LIN {X 0,Y 573.255,Z 289.769,A -85,B 0,C 180,E1 -2241.895,E2 -2241.895} C_VEL
LIN {X 0,Y 573.193,Z 298.434,A -85,B 0,C 180,E1 -2242.603,E2 -2242.603} C_VEL
LIN {X 0,Y 573.151,Z 305.582,A -85,B 0,C 180,E1 -2243.326,E2 -2243.326} C_VEL
LIN {X 0,Y 573.113,Z 312.436,A -85,B 0,C 180,E1 -2244.194,E2 -2244.194} C_VEL
LIN {X 0,Y 572.995,Z 317.989,A -85,B 0,C 180,E1 -2245.075,E2 -2245.075} C_VEL
LIN {X 0,Y 573.036,Z 323.15,A -85,B 0,C 180,E1 -2246.132,E2 -2246.132} C_VEL
LIN {X 0,Y 572.99,Z 325.788,A -85,B 0,C 180,E1 -2246.836,E2 -2246.836} C_VEL
LIN {X 0,Y 572.94,Z 328.683,A -85,B 0,C 180,E1 -2247.891,E2 -2247.891} C_VEL
LIN {X 0,Y 572.944,Z 329.933,A -85,B 0,C 180,E1 -2248.594,E2 -2248.594} C_VEL
LIN {X 0,Y 572.937,Z 330.709,A -85,B 0,C 180,E1 -2249.297,E2 -2249.297} C_VEL
LIN {X 0,Y 572.935,Z 331,A -85,B 0,C 180,E1 -2250,E2 -2250} C_VEL
LIN {X 0,Y 572.937,Z 330.708,A -85,B 0,C 180,E1 -2250.703,E2 -2250.703} C_VEL
LIN {X 0,Y 572.944,Z 329.932,A -85,B 0,C 180,E1 -2251.406,E2 -2251.406} C_VEL
LIN {X 0,Y 572.94,Z 328.681,A -85,B 0,C 180,E1 -2252.109,E2 -2252.109} C_VEL
LIN {X 0,Y 572.99,Z 325.787,A -85,B 0,C 180,E1 -2253.164,E2 -2253.164} C_VEL
LIN {X 0,Y 573.036,Z 323.148,A -85,B 0,C 180,E1 -2253.868,E2 -2253.868} C_VEL
LIN {X 0,Y 572.995,Z 317.985,A -85,B 0,C 180,E1 -2254.926,E2 -2254.926} C_VEL
LIN {X 0,Y 573.138,Z 311.184,A -85,B 0,C 180,E1 -2255.983,E2 -2255.983} C_VEL
LIN {X 0,Y 573.163,Z 303.801,A -85,B 0,C 180,E1 -2256.86,E2 -2256.86} C_VEL
LIN {X 0,Y 573.216,Z 296.401,A -85,B 0,C 180,E1 -2257.574,E2 -2257.574} C_VEL
LIN {X 0,Y 573.277,Z 288.538,A -85,B 0,C 180,E1 -2258.194,E2 -2258.194} C_VEL
LIN {X 0,Y 573.4,Z 278.724,A -85,B 0,C 180,E1 -2258.813,E2 -2258.813} C_VEL
LIN {X 0,Y 573.468,Z 267.301,A -85,B 0,C 180,E1 -2259.345,E2 -2259.345} C_VEL
LIN {X 0,Y 573.529,Z 257.24,A -85,B 0,C 180,E1 -2259.678,E2 -2259.678} C_VEL
LIN {X 0,Y 573.594,Z 248.431,A -85,B 0,C 180,E1 -2259.877,E2 -2259.877} C_VEL
LIN {X 0,Y 573.656,Z 186.16,A -85,B 0,C 180,E1 -2260.674,E2 -2260.674} C_VEL
LIN {X 0,Y 573.48,Z 173.915,A -85,B 0,C 180,E1 -2260.831,E2 -2260.831} C_VEL
LIN {X 0,Y 573.188,Z 171.334,A -85,B 0,C 180,E1 -2260.895,E2 -2260.895} C_VEL
LIN {X 0,Y 573.23,Z 164.43,A -85,B 0,C 180,E1 -2262.03,E2 -2262.03} C_VEL
LIN {X 0,Y 573.33,Z 147.689,A -85,B 0,C 180,E1 -2264.917,E2 -2264.917} C_VEL
LIN {X 0,Y 573.51,Z 129.794,A -85,B 0,C 180,E1 -2268.025,E2 -2268.025} C_VEL
LIN {X 0,Y 573.612,Z 115.014,A -85,B 0,C 180,E1 -2270.625,E2 -2270.625} C_VEL
LIN {X 0,Y 573.276,Z 111.928,A -85,B 0,C 180,E1 -2271.23,E2 -2271.23} C_VEL
LIN {X 0,Y 573.222,Z 111.88,A -85,B 0,C 180,E1 -2273.866,E2 -2273.866} C_VEL
LIN {X 0,Y 573.236,Z 111.897,A -85,B 0,C 180,E1 -2276.492,E2 -2276.492} C_VEL
LIN {X 0,Y 573.239,Z 111.894,A -85,B 0,C 180,E1 -2278.564,E2 -2278.564} C_VEL
LIN {X 0,Y 573.225,Z 111.89,A -85,B 0,C 180,E1 -2280.993,E2 -2280.993} C_VEL
LIN {X 0,Y 573.263,Z 111.885,A -85,B 0,C 180,E1 -2283.524,E2 -2283.524} C_VEL
LIN {X 0,Y 573.215,Z 111.899,A -85,B 0,C 180,E1 -2286.052,E2 -2286.052} C_VEL
LIN {X 0,Y 573.242,Z 111.888,A -85,B 0,C 180,E1 -2288.702,E2 -2288.702} C_VEL
LIN {X 0,Y 573.23,Z 111.893,A -85,B 0,C 180,E1 -2291.593,E2 -2291.593} C_VEL
LIN {X 0,Y 573.222,Z 111.891,A -85,B 0,C 180,E1 -2294.335,E2 -2294.335} C_VEL
LIN {X 0,Y 573.241,Z 111.891,A -85,B 0,C 180,E1 -2297.359,E2 -2297.359} C_VEL
LIN {X 0,Y 573.24,Z 111.887,A -85,B 0,C 180,E1 -2300.392,E2 -2300.392} C_VEL
LIN {X 0,Y 573.256,Z 111.889,A -85,B 0,C 180,E1 -2303.078,E2 -2303.078} C_VEL
LIN {X 0,Y 573.268,Z 111.888,A -85,B 0,C 180,E1 -2305.671,E2 -2305.671} C_VEL
LIN {X 0,Y 573.241,Z 111.887,A -85,B 0,C 180,E1 -2308.185,E2 -2308.185} C_VEL
LIN {X 0,Y 573.265,Z 111.886,A -85,B 0,C 180,E1 -2310.634,E2 -2310.634} C_VEL
LIN {X 0,Y 573.251,Z 111.894,A -85,B 0,C 180,E1 -2313.024,E2 -2313.024} C_VEL
LIN {X 0,Y 573.275,Z 111.886,A -85,B 0,C 180,E1 -2315.366,E2 -2315.366} C_VEL
LIN {X 0,Y 573.23,Z 111.891,A -85,B 0,C 180,E1 -2318.419,E2 -2318.419} C_VEL
LIN {X 0,Y 573.28,Z 111.891,A -85,B 0,C 180,E1 -2320.728,E2 -2320.728} C_VEL
LIN {X 0,Y 573.252,Z 111.885,A -85,B 0,C 180,E1 -2323.622,E2 -2323.622} C_VEL
LIN {X 0,Y 573.274,Z 111.883,A -85,B 0,C 180,E1 -2325.807,E2 -2325.807} C_VEL
LIN {X 0,Y 573.265,Z 111.889,A -85,B 0,C 180,E1 -2328.745,E2 -2328.745} C_VEL
LIN {X 0,Y 573.285,Z 111.882,A -85,B 0,C 180,E1 -2331.541,E2 -2331.541} C_VEL
LIN {X 0,Y 573.289,Z 111.889,A -85,B 0,C 180,E1 -2334.372,E2 -2334.372} C_VEL
LIN {X 0,Y 573.311,Z 111.884,A -85,B 0,C 180,E1 -2337.893,E2 -2337.893} C_VEL
LIN {X 0,Y 573.333,Z 111.876,A -85,B 0,C 180,E1 -2340.702,E2 -2340.702} C_VEL
LIN {X 0,Y 573.304,Z 111.879,A -85,B 0,C 180,E1 -2342.811,E2 -2342.811} C_VEL
LIN {X 0,Y 573.289,Z 111.887,A -85,B 0,C 180,E1 -2345.628,E2 -2345.628} C_VEL
LIN {X 0,Y 573.286,Z 111.882,A -85,B 0,C 180,E1 -2348.46,E2 -2348.46} C_VEL
LIN {X 0,Y 573.274,Z 111.887,A -85,B 0,C 180,E1 -2351.312,E2 -2351.312} C_VEL
LIN {X 0,Y 573.283,Z 111.882,A -85,B 0,C 180,E1 -2354.424,E2 -2354.424} C_VEL
LIN {X 0,Y 573.26,Z 111.889,A -85,B 0,C 180,E1 -2357.112,E2 -2357.112} C_VEL
LIN {X 0,Y 573.244,Z 111.887,A -85,B 0,C 180,E1 -2360.077,E2 -2360.077} C_VEL
LIN {X 0,Y 573.237,Z 111.887,A -85,B 0,C 180,E1 -2362.338,E2 -2362.338} C_VEL
LIN {X 0,Y 573.25,Z 111.886,A -85,B 0,C 180,E1 -2364.384,E2 -2364.384} C_VEL
LIN {X 0,Y 572.625,Z 111.971,A -85,B 0,C 180,E1 -2364.97,E2 -2364.97} C_VEL
LIN {X 0,Y 569.784,Z 112.326,A -85,B 0,C 180,E1 -2365.922,E2 -2365.922} C_VEL
LIN {X 0,Y 567.351,Z 112.629,A -85,B 0,C 180,E1 -2366.687,E2 -2366.687} C_VEL
LIN {X 0,Y 566.295,Z 112.758,A -85,B 0,C 180,E1 -2367.278,E2 -2367.278} C_VEL
LIN {X 0,Y 566.205,Z 112.766,A -85,B 0,C 180,E1 -2367.479,E2 -2367.479} C_VEL
LIN {X 0,Y 566.203,Z 112.764,A -85,B 0,C 180,E1 -2369.769,E2 -2369.769} C_VEL
LIN {X 0,Y 566.204,Z 112.767,A -85,B 0,C 180,E1 -2372.43,E2 -2372.43} C_VEL
LIN {X 0,Y 566.205,Z 112.769,A -85,B 0,C 180,E1 -2374.993,E2 -2374.993} C_VEL
LIN {X 0,Y 566.198,Z 112.764,A -85,B 0,C 180,E1 -2377.461,E2 -2377.461} C_VEL
LIN {X 0,Y 566.209,Z 112.767,A -85,B 0,C 180,E1 -2380.199,E2 -2380.199} C_VEL
LIN {X 0,Y 566.202,Z 112.765,A -85,B 0,C 180,E1 -2383.054,E2 -2383.054} C_VEL
LIN {X 0,Y 566.195,Z 112.769,A -85,B 0,C 180,E1 -2386.049,E2 -2386.049} C_VEL
LIN {X 0,Y 566.205,Z 112.763,A -85,B 0,C 180,E1 -2389.215,E2 -2389.215} C_VEL
LIN {X 0,Y 566.187,Z 112.768,A -85,B 0,C 180,E1 -2391.637,E2 -2391.637} C_VEL
LIN {X 0,Y 566.195,Z 112.77,A -85,B 0,C 180,E1 -2394.31,E2 -2394.31} C_VEL
LIN {X 0,Y 566.206,Z 112.763,A -85,B 0,C 180,E1 -2396.897,E2 -2396.897} C_VEL
LIN {X 0,Y 566.183,Z 112.769,A -85,B 0,C 180,E1 -2399.407,E2 -2399.407} C_VEL
LIN {X 0,Y 566.214,Z 112.77,A -85,B 0,C 180,E1 -2401.857,E2 -2401.857} C_VEL
LIN {X 0,Y 566.214,Z 112.764,A -85,B 0,C 180,E1 -2404.251,E2 -2404.251} C_VEL
LIN {X 0,Y 566.171,Z 112.768,A -85,B 0,C 180,E1 -2406.719,E2 -2406.719} C_VEL
LIN {X 0,Y 566.21,Z 112.771,A -85,B 0,C 180,E1 -2409.663,E2 -2409.663} C_VEL
LIN {X 0,Y 566.266,Z 112.994,A -85,B 0,C 180,E1 -2411.1,E2 -2411.1} C_VEL
LIN {X 0,Y 566.314,Z 124.262,A -85,B 0,C 180,E1 -2413.415,E2 -2413.415} C_VEL
LIN {X 0,Y 566.184,Z 138.786,A -85,B 0,C 180,E1 -2416.358,E2 -2416.358} C_VEL
LIN {X 0,Y 566.08,Z 152.209,A -85,B 0,C 180,E1 -2419.011,E2 -2419.011} C_VEL
LIN {X 0,Y 566.347,Z 154.505,A -85,B 0,C 180,E1 -2419.084,E2 -2419.084} C_VEL
LIN {X 0,Y 566.716,Z 161.739,A -85,B 0,C 180,E1 -2419.182,E2 -2419.182} C_VEL
LIN {X 0,Y 566.594,Z 228.447,A -85,B 0,C 180,E1 -2420.045,E2 -2420.045} C_VEL
LIN {X 0,Y 566.527,Z 238.091,A -85,B 0,C 180,E1 -2420.269,E2 -2420.269} C_VEL
LIN {X 0,Y 566.442,Z 249.61,A -85,B 0,C 180,E1 -2420.673,E2 -2420.673} C_VEL
LIN {X 0,Y 566.309,Z 259.464,A -85,B 0,C 180,E1 -2421.166,E2 -2421.166} C_VEL
LIN {X 0,Y 566.261,Z 267.916,A -85,B 0,C 180,E1 -2421.704,E2 -2421.704} C_VEL
LIN {X 0,Y 566.17,Z 275.886,A -85,B 0,C 180,E1 -2422.331,E2 -2422.331} C_VEL
LIN {X 0,Y 566.097,Z 282.681,A -85,B 0,C 180,E1 -2422.981,E2 -2422.981} C_VEL
LIN {X 0,Y 566.063,Z 287.999,A -85,B 0,C 180,E1 -2423.584,E2 -2423.584} C_VEL
LIN {X 0,Y 566.025,Z 293.312,A -85,B 0,C 180,E1 -2424.299,E2 -2424.299} C_VEL
LIN {X 0,Y 565.917,Z 297.747,A -85,B 0,C 180,E1 -2425.013,E2 -2425.013} C_VEL
LIN {X 0,Y 565.961,Z 301.44,A -85,B 0,C 180,E1 -2425.727,E2 -2425.727} C_VEL
LIN {X 0,Y 565.914,Z 305.642,A -85,B 0,C 180,E1 -2426.796,E2 -2426.796} C_VEL
LIN {X 0,Y 565.841,Z 308.582,A -85,B 0,C 180,E1 -2427.864,E2 -2427.864} C_VEL
LIN {X 0,Y 565.843,Z 309.872,A -85,B 0,C 180,E1 -2428.576,E2 -2428.576} C_VEL
LIN {X 0,Y 565.837,Z 310.688,A -85,B 0,C 180,E1 -2429.288,E2 -2429.288} C_VEL
LIN {X 0,Y 565.837,Z 310.996,A -85,B 0,C 180,E1 -2430,E2 -2430} C_VEL
LIN {X 0,Y 565.838,Z 310.729,A -85,B 0,C 180,E1 -2430.711,E2 -2430.711} C_VEL
LIN {X 0,Y 565.845,Z 309.993,A -85,B 0,C 180,E1 -2431.423,E2 -2431.423} C_VEL
LIN {X 0,Y 565.841,Z 308.788,A -85,B 0,C 180,E1 -2432.135,E2 -2432.135} C_VEL
LIN {X 0,Y 565.913,Z 305.935,A -85,B 0,C 180,E1 -2433.203,E2 -2433.203} C_VEL
LIN {X 0,Y 565.963,Z 301.824,A -85,B 0,C 180,E1 -2434.273,E2 -2434.273} C_VEL
LIN {X 0,Y 565.946,Z 296.247,A -85,B 0,C 180,E1 -2435.344,E2 -2435.344} C_VEL
LIN {X 0,Y 566.077,Z 290.136,A -85,B 0,C 180,E1 -2436.236,E2 -2436.236} C_VEL
LIN {X 0,Y 566.098,Z 284.166,A -85,B 0,C 180,E1 -2436.953,E2 -2436.953} C_VEL
LIN {X 0,Y 566.15,Z 276.915,A -85,B 0,C 180,E1 -2437.669,E2 -2437.669} C_VEL
LIN {X 0,Y 566.24,Z 269.155,A -85,B 0,C 180,E1 -2438.296,E2 -2438.296} C_VEL
LIN {X 0,Y 566.301,Z 260.976,A -85,B 0,C 180,E1 -2438.834,E2 -2438.834} C_VEL
LIN {X 0,Y 566.441,Z 250.583,A -85,B 0,C 180,E1 -2439.372,E2 -2439.372} C_VEL
LIN {X 0,Y 566.545,Z 238.933,A -85,B 0,C 180,E1 -2439.798,E2 -2439.798} C_VEL
LIN {X 0,Y 566.613,Z 228.456,A -85,B 0,C 180,E1 -2440.045,E2 -2440.045} C_VEL
LIN {X 0,Y 566.586,Z 156.361,A -85,B 0,C 180,E1 -2440.978,E2 -2440.978} C_VEL
LIN {X 0,Y 566.146,Z 152.501,A -85,B 0,C 180,E1 -2441.057,E2 -2441.057} C_VEL
LIN {X 0,Y 566.067,Z 151.18,A -85,B 0,C 180,E1 -2441.238,E2 -2441.238} C_VEL
LIN {X 0,Y 566.182,Z 137.43,A -85,B 0,C 180,E1 -2444.008,E2 -2444.008} C_VEL
LIN {X 0,Y 566.314,Z 123.312,A -85,B 0,C 180,E1 -2446.867,E2 -2446.867} C_VEL
LIN {X 0,Y 566.276,Z 112.863,A -85,B 0,C 180,E1 -2449.032,E2 -2449.032} C_VEL
LIN {X 0,Y 566.193,Z 112.767,A -85,B 0,C 180,E1 -2451.862,E2 -2451.862} C_VEL
LIN {X 0,Y 566.219,Z 112.763,A -85,B 0,C 180,E1 -2455.03,E2 -2455.03} C_VEL
LIN {X 0,Y 566.212,Z 112.762,A -85,B 0,C 180,E1 -2457.339,E2 -2457.339} C_VEL
LIN {X 0,Y 566.201,Z 112.766,A -85,B 0,C 180,E1 -2459.769,E2 -2459.769} C_VEL
LIN {X 0,Y 566.204,Z 112.769,A -85,B 0,C 180,E1 -2462.43,E2 -2462.43} C_VEL
LIN {X 0,Y 566.203,Z 112.764,A -85,B 0,C 180,E1 -2464.993,E2 -2464.993} C_VEL
LIN {X 0,Y 566.196,Z 112.767,A -85,B 0,C 180,E1 -2467.461,E2 -2467.461} C_VEL
LIN {X 0,Y 566.207,Z 112.768,A -85,B 0,C 180,E1 -2470.199,E2 -2470.199} C_VEL
LIN {X 0,Y 566.199,Z 112.765,A -85,B 0,C 180,E1 -2473.054,E2 -2473.054} C_VEL
LIN {X 0,Y 566.197,Z 112.768,A -85,B 0,C 180,E1 -2476.048,E2 -2476.048} C_VEL
LIN {X 0,Y 566.178,Z 112.768,A -85,B 0,C 180,E1 -2478.861,E2 -2478.861} C_VEL
LIN {X 0,Y 566.185,Z 112.772,A -85,B 0,C 180,E1 -2481.637,E2 -2481.637} C_VEL
LIN {X 0,Y 566.196,Z 112.764,A -85,B 0,C 180,E1 -2484.31,E2 -2484.31} C_VEL
LIN {X 0,Y 566.219,Z 112.766,A -85,B 0,C 180,E1 -2486.898,E2 -2486.898} C_VEL
LIN {X 0,Y 566.181,Z 112.772,A -85,B 0,C 180,E1 -2489.407,E2 -2489.407} C_VEL
LIN {X 0,Y 566.211,Z 112.763,A -85,B 0,C 180,E1 -2491.857,E2 -2491.857} C_VEL
LIN {X 0,Y 566.212,Z 112.763,A -85,B 0,C 180,E1 -2494.251,E2 -2494.251} C_VEL
LIN {X 0,Y 566.172,Z 112.775,A -85,B 0,C 180,E1 -2496.718,E2 -2496.718} C_VEL
LIN {X 0,Y 566.213,Z 112.762,A -85,B 0,C 180,E1 -2499.663,E2 -2499.663} C_VEL
LIN {X 0,Y 566.2,Z 112.773,A -85,B 0,C 180,E1 -2502.668,E2 -2502.668} C_VEL
LIN {X 0,Y 566.233,Z 112.76,A -85,B 0,C 180,E1 -2505.627,E2 -2505.627} C_VEL
LIN {X 0,Y 566.234,Z 112.765,A -85,B 0,C 180,E1 -2508.675,E2 -2508.675} C_VEL
LIN {X 0,Y 566.227,Z 112.761,A -85,B 0,C 180,E1 -2511.434,E2 -2511.434} C_VEL
LIN {X 0,Y 566.259,Z 112.764,A -85,B 0,C 180,E1 -2514.302,E2 -2514.302} C_VEL
LIN {X 0,Y 566.284,Z 112.76,A -85,B 0,C 180,E1 -2517.866,E2 -2517.866} C_VEL
LIN {X 0,Y 566.301,Z 112.752,A -85,B 0,C 180,E1 -2520.711,E2 -2520.711} C_VEL
LIN {X 0,Y 566.27,Z 112.755,A -85,B 0,C 180,E1 -2522.845,E2 -2522.845} C_VEL
LIN {X 0,Y 566.258,Z 112.765,A -85,B 0,C 180,E1 -2525.698,E2 -2525.698} C_VEL
LIN {X 0,Y 566.227,Z 112.761,A -85,B 0,C 180,E1 -2528.566,E2 -2528.566} C_VEL
LIN {X 0,Y 566.241,Z 112.767,A -85,B 0,C 180,E1 -2531.454,E2 -2531.454} C_VEL
LIN {X 0,Y 566.233,Z 112.76,A -85,B 0,C 180,E1 -2534.507,E2 -2534.507} C_VEL
LIN {X 0,Y 566.199,Z 112.773,A -85,B 0,C 180,E1 -2537.332,E2 -2537.332} C_VEL
LIN {X 0,Y 566.213,Z 112.762,A -85,B 0,C 180,E1 -2540.337,E2 -2540.337} C_VEL
LIN {X 0,Y 566.168,Z 112.774,A -85,B 0,C 180,E1 -2543.281,E2 -2543.281} C_VEL
LIN {X 0,Y 566.211,Z 112.763,A -85,B 0,C 180,E1 -2545.749,E2 -2545.749} C_VEL
LIN {X 0,Y 566.201,Z 112.765,A -85,B 0,C 180,E1 -2548.202,E2 -2548.202} C_VEL
LIN {X 0,Y 566.19,Z 112.77,A -85,B 0,C 180,E1 -2551.077,E2 -2551.077} C_VEL
LIN {X 0,Y 566.21,Z 112.763,A -85,B 0,C 180,E1 -2553.734,E2 -2553.734} C_VEL
LIN {X 0,Y 566.209,Z 112.773,A -85,B 0,C 180,E1 -2556.569,E2 -2556.569} C_VEL
LIN {X 0,Y 566.214,Z 112.763,A -85,B 0,C 180,E1 -2559.686,E2 -2559.686} C_VEL
LIN {X 0,Y 566.209,Z 112.768,A -85,B 0,C 180,E1 -2562.088,E2 -2562.088} C_VEL
LIN {X 0,Y 566.167,Z 112.768,A -85,B 0,C 180,E1 -2565.037,E2 -2565.037} C_VEL
LIN {X 0,Y 566.207,Z 112.769,A -85,B 0,C 180,E1 -2567.912,E2 -2567.912} C_VEL
LIN {X 0,Y 566.213,Z 112.763,A -85,B 0,C 180,E1 -2570.727,E2 -2570.727} C_VEL
LIN {X 0,Y 566.201,Z 112.771,A -85,B 0,C 180,E1 -2573.786,E2 -2573.786} C_VEL
LIN {X 0,Y 566.197,Z 112.767,A -85,B 0,C 180,E1 -2576.268,E2 -2576.268} C_VEL
LIN {X 0,Y 566.189,Z 112.766,A -85,B 0,C 180,E1 -2578.924,E2 -2578.924} C_VEL
LIN {X 0,Y 566.211,Z 112.768,A -85,B 0,C 180,E1 -2581.858,E2 -2581.858} C_VEL
LIN {X 0,Y 566.208,Z 112.764,A -85,B 0,C 180,E1 -2584.251,E2 -2584.251} C_VEL
LIN {X 0,Y 566.167,Z 112.761,A -85,B 0,C 180,E1 -2586.72,E2 -2586.72} C_VEL
LIN {X 0,Y 566.24,Z 112.918,A -85,B 0,C 180,E1 -2588.725,E2 -2588.725} C_VEL
LIN {X 0,Y 566.614,Z 117.013,A -85,B 0,C 180,E1 -2589.489,E2 -2589.489} C_VEL
LIN {X 0,Y 566.45,Z 133.899,A -85,B 0,C 180,E1 -2592.49,E2 -2592.49} C_VEL
LIN {X 0,Y 566.288,Z 149.636,A -85,B 0,C 180,E1 -2595.247,E2 -2595.247} C_VEL
LIN {X 0,Y 566.178,Z 166.525,A -85,B 0,C 180,E1 -2598.182,E2 -2598.182} C_VEL
LIN {X 0,Y 566.125,Z 171.19,A -85,B 0,C 180,E1 -2598.956,E2 -2598.956} C_VEL
LIN {X 0,Y 566.38,Z 173.554,A -85,B 0,C 180,E1 -2599.027,E2 -2599.027} C_VEL
LIN {X 0,Y 566.695,Z 184.814,A -85,B 0,C 180,E1 -2599.176,E2 -2599.176} C_VEL
LIN {X 0,Y 566.59,Z 247.151,A -85,B 0,C 180,E1 -2599.977,E2 -2599.977} C_VEL
LIN {X 0,Y 566.518,Z 256.418,A -85,B 0,C 180,E1 -2600.179,E2 -2600.179} C_VEL
LIN {X 0,Y 566.472,Z 264.89,A -85,B 0,C 180,E1 -2600.448,E2 -2600.448} C_VEL
LIN {X 0,Y 566.415,Z 273.394,A -85,B 0,C 180,E1 -2600.808,E2 -2600.808} C_VEL
LIN {X 0,Y 566.328,Z 281.727,A -85,B 0,C 180,E1 -2601.256,E2 -2601.256} C_VEL
LIN {X 0,Y 566.211,Z 289.765,A -85,B 0,C 180,E1 -2601.794,E2 -2601.794} C_VEL
LIN {X 0,Y 566.127,Z 298.434,A -85,B 0,C 180,E1 -2602.51,E2 -2602.51} C_VEL
LIN {X 0,Y 566.091,Z 306.878,A -85,B 0,C 180,E1 -2603.398,E2 -2603.398} C_VEL
LIN {X 0,Y 566.057,Z 312.437,A -85,B 0,C 180,E1 -2604.121,E2 -2604.121} C_VEL
LIN {X 0,Y 565.906,Z 317.99,A -85,B 0,C 180,E1 -2605.013,E2 -2605.013} C_VEL
LIN {X 0,Y 565.943,Z 323.15,A -85,B 0,C 180,E1 -2606.084,E2 -2606.084} C_VEL
LIN {X 0,Y 565.88,Z 326.937,A -85,B 0,C 180,E1 -2607.153,E2 -2607.153} C_VEL
LIN {X 0,Y 565.841,Z 328.682,A -85,B 0,C 180,E1 -2607.865,E2 -2607.865} C_VEL
LIN {X 0,Y 565.844,Z 329.932,A -85,B 0,C 180,E1 -2608.577,E2 -2608.577} C_VEL
LIN {X 0,Y 565.837,Z 330.708,A -85,B 0,C 180,E1 -2609.289,E2 -2609.289} C_VEL
LIN {X 0,Y 565.836,Z 331,A -85,B 0,C 180,E1 -2610,E2 -2610} C_VEL
LIN {X 0,Y 565.837,Z 330.707,A -85,B 0,C 180,E1 -2610.712,E2 -2610.712} C_VEL
LIN {X 0,Y 565.844,Z 329.931,A -85,B 0,C 180,E1 -2611.424,E2 -2611.424} C_VEL
LIN {X 0,Y 565.841,Z 328.681,A -85,B 0,C 180,E1 -2612.136,E2 -2612.136} C_VEL
LIN {X 0,Y 565.912,Z 325.786,A -85,B 0,C 180,E1 -2613.204,E2 -2613.204} C_VEL
LIN {X 0,Y 565.944,Z 323.148,A -85,B 0,C 180,E1 -2613.917,E2 -2613.917} C_VEL
LIN {X 0,Y 565.906,Z 317.985,A -85,B 0,C 180,E1 -2614.987,E2 -2614.987} C_VEL
LIN {X 0,Y 566.082,Z 311.182,A -85,B 0,C 180,E1 -2616.058,E2 -2616.058} C_VEL
LIN {X 0,Y 566.091,Z 304.175,A -85,B 0,C 180,E1 -2616.907,E2 -2616.907} C_VEL
LIN {X 0,Y 566.149,Z 296.398,A -85,B 0,C 180,E1 -2617.669,E2 -2617.669} C_VEL
LIN {X 0,Y 566.239,Z 288.534,A -85,B 0,C 180,E1 -2618.296,E2 -2618.296} C_VEL
LIN {X 0,Y 566.333,Z 280.221,A -85,B 0,C 180,E1 -2618.834,E2 -2618.834} C_VEL
LIN {X 0,Y 566.46,Z 269.607,A -85,B 0,C 180,E1 -2619.372,E2 -2619.372} C_VEL
LIN {X 0,Y 566.54,Z 258.07,A -85,B 0,C 180,E1 -2619.776,E2 -2619.776} C_VEL
LIN {X 0,Y 566.62,Z 248.43,A -85,B 0,C 180,E1 -2620,E2 -2620} C_VEL
LIN {X 0,Y 566.703,Z 185.955,A -85,B 0,C 180,E1 -2620.81,E2 -2620.81} C_VEL
LIN {X 0,Y 566.451,Z 174.275,A -85,B 0,C 180,E1 -2620.962,E2 -2620.962} C_VEL
LIN {X 0,Y 566.152,Z 171.448,A -85,B 0,C 180,E1 -2621.025,E2 -2621.025} C_VEL
LIN {X 0,Y 566.13,Z 168.615,A -85,B 0,C 180,E1 -2621.457,E2 -2621.457} C_VEL
LIN {X 0,Y 566.273,Z 150.965,A -85,B 0,C 180,E1 -2624.521,E2 -2624.521} C_VEL
LIN {X 0,Y 566.437,Z 134.948,A -85,B 0,C 180,E1 -2627.324,E2 -2627.324} C_VEL
LIN {X 0,Y 566.592,Z 118.066,A -85,B 0,C 180,E1 -2630.323,E2 -2630.323} C_VEL
LIN {X 0,Y 566.297,Z 113.186,A -85,B 0,C 180,E1 -2631.214,E2 -2631.214} C_VEL
LIN {X 0,Y 566.215,Z 112.77,A -85,B 0,C 180,E1 -2631.422,E2 -2631.422} C_VEL
LIN {X 0,Y 566.193,Z 112.759,A -85,B 0,C 180,E1 -2634.181,E2 -2634.181} C_VEL
LIN {X 0,Y 566.208,Z 112.769,A -85,B 0,C 180,E1 -2636.659,E2 -2636.659} C_VEL
LIN {X 0,Y 566.192,Z 112.767,A -85,B 0,C 180,E1 -2638.953,E2 -2638.953} C_VEL
LIN {X 0,Y 566.193,Z 112.765,A -85,B 0,C 180,E1 -2641.422,E2 -2641.422} C_VEL
LIN {X 0,Y 566.21,Z 112.769,A -85,B 0,C 180,E1 -2643.956,E2 -2643.956} C_VEL
LIN {X 0,Y 566.2,Z 112.766,A -85,B 0,C 180,E1 -2646.57,E2 -2646.57} C_VEL
LIN {X 0,Y 566.215,Z 112.767,A -85,B 0,C 180,E1 -2649.686,E2 -2649.686} C_VEL
LIN {X 0,Y 566.201,Z 112.764,A -85,B 0,C 180,E1 -2652.917,E2 -2652.917} C_VEL
LIN {X 0,Y 566.194,Z 112.769,A -85,B 0,C 180,E1 -2656.049,E2 -2656.049} C_VEL
LIN {X 0,Y 566.179,Z 112.767,A -85,B 0,C 180,E1 -2658.861,E2 -2658.861} C_VEL
LIN {X 0,Y 566.186,Z 112.773,A -85,B 0,C 180,E1 -2661.637,E2 -2661.637} C_VEL
LIN {X 0,Y 566.197,Z 112.764,A -85,B 0,C 180,E1 -2664.31,E2 -2664.31} C_VEL
LIN {X 0,Y 566.221,Z 112.765,A -85,B 0,C 180,E1 -2666.898,E2 -2666.898} C_VEL
LIN {X 0,Y 566.182,Z 112.773,A -85,B 0,C 180,E1 -2669.407,E2 -2669.407} C_VEL
LIN {X 0,Y 566.213,Z 112.763,A -85,B 0,C 180,E1 -2671.858,E2 -2671.858} C_VEL
LIN {X 0,Y 566.21,Z 112.763,A -85,B 0,C 180,E1 -2674.251,E2 -2674.251} C_VEL
LIN {X 0,Y 566.17,Z 112.773,A -85,B 0,C 180,E1 -2676.719,E2 -2676.719} C_VEL
LIN {X 0,Y 566.215,Z 112.762,A -85,B 0,C 180,E1 -2679.663,E2 -2679.663} C_VEL
LIN {X 0,Y 566.201,Z 112.773,A -85,B 0,C 180,E1 -2682.668,E2 -2682.668} C_VEL
LIN {X 0,Y 566.235,Z 112.759,A -85,B 0,C 180,E1 -2685.627,E2 -2685.627} C_VEL
LIN {X 0,Y 566.236,Z 112.766,A -85,B 0,C 180,E1 -2688.675,E2 -2688.675} C_VEL
LIN {X 0,Y 566.229,Z 112.76,A -85,B 0,C 180,E1 -2691.434,E2 -2691.434} C_VEL
LIN {X 0,Y 566.257,Z 112.766,A -85,B 0,C 180,E1 -2694.302,E2 -2694.302} C_VEL
LIN {X 0,Y 566.282,Z 112.759,A -85,B 0,C 180,E1 -2697.866,E2 -2697.866} C_VEL
LIN {X 0,Y 566.303,Z 112.752,A -85,B 0,C 180,E1 -2700.711,E2 -2700.711} C_VEL
LIN {X 0,Y 566.27,Z 112.755,A -85,B 0,C 180,E1 -2702.846,E2 -2702.846} C_VEL
LIN {X 0,Y 566.258,Z 112.764,A -85,B 0,C 180,E1 -2705.698,E2 -2705.698} C_VEL
LIN {X 0,Y 566.229,Z 112.761,A -85,B 0,C 180,E1 -2708.566,E2 -2708.566} C_VEL
LIN {X 0,Y 566.244,Z 112.765,A -85,B 0,C 180,E1 -2711.454,E2 -2711.454} C_VEL
LIN {X 0,Y 566.236,Z 112.759,A -85,B 0,C 180,E1 -2714.506,E2 -2714.506} C_VEL
LIN {X 0,Y 566.202,Z 112.772,A -85,B 0,C 180,E1 -2717.332,E2 -2717.332} C_VEL
LIN {X 0,Y 566.209,Z 112.763,A -85,B 0,C 180,E1 -2720.337,E2 -2720.337} C_VEL
LIN {X 0,Y 566.171,Z 112.776,A -85,B 0,C 180,E1 -2723.281,E2 -2723.281} C_VEL
LIN {X 0,Y 566.214,Z 112.763,A -85,B 0,C 180,E1 -2725.749,E2 -2725.749} C_VEL
LIN {X 0,Y 566.205,Z 112.766,A -85,B 0,C 180,E1 -2727.479,E2 -2727.479} C_VEL
LIN {X 0,Y 565.525,Z 112.85,A -85,B 0,C 180,E1 -2728.072,E2 -2728.072} C_VEL
LIN {X 0,Y 562.659,Z 113.214,A -85,B 0,C 180,E1 -2729.036,E2 -2729.036} C_VEL
LIN {X 0,Y 560.249,Z 113.509,A -85,B 0,C 180,E1 -2729.812,E2 -2729.812} C_VEL
LIN {X 0,Y 559.222,Z 113.635,A -85,B 0,C 180,E1 -2730.41,E2 -2730.41} C_VEL
LIN {X 0,Y 559.141,Z 113.646,A -85,B 0,C 180,E1 -2730.613,E2 -2730.613} C_VEL
LIN {X 0,Y 559.164,Z 113.641,A -85,B 0,C 180,E1 -2733.575,E2 -2733.575} C_VEL
LIN {X 0,Y 559.163,Z 113.646,A -85,B 0,C 180,E1 -2736.447,E2 -2736.447} C_VEL
LIN {X 0,Y 559.176,Z 113.643,A -85,B 0,C 180,E1 -2738.934,E2 -2738.934} C_VEL
LIN {X 0,Y 559.164,Z 113.641,A -85,B 0,C 180,E1 -2741.77,E2 -2741.77} C_VEL
LIN {X 0,Y 559.133,Z 113.648,A -85,B 0,C 180,E1 -2744.74,E2 -2744.74} C_VEL
LIN {X 0,Y 559.159,Z 113.641,A -85,B 0,C 180,E1 -2747.256,E2 -2747.256} C_VEL
LIN {X 0,Y 559.181,Z 113.647,A -85,B 0,C 180,E1 -2750.134,E2 -2750.134} C_VEL
LIN {X 0,Y 559.145,Z 113.643,A -85,B 0,C 180,E1 -2752.892,E2 -2752.892} C_VEL
LIN {X 0,Y 559.149,Z 113.645,A -85,B 0,C 180,E1 -2755.555,E2 -2755.555} C_VEL
LIN {X 0,Y 559.167,Z 113.645,A -85,B 0,C 180,E1 -2758.137,E2 -2758.137} C_VEL
LIN {X 0,Y 559.144,Z 113.643,A -85,B 0,C 180,E1 -2760.646,E2 -2760.646} C_VEL
LIN {X 0,Y 559.173,Z 113.641,A -85,B 0,C 180,E1 -2763.173,E2 -2763.173} C_VEL
LIN {X 0,Y 559.158,Z 113.649,A -85,B 0,C 180,E1 -2765.495,E2 -2765.495} C_VEL
LIN {X 0,Y 559.174,Z 113.641,A -85,B 0,C 180,E1 -2768.624,E2 -2768.624} C_VEL
LIN {X 0,Y 559.225,Z 113.817,A -85,B 0,C 180,E1 -2771.023,E2 -2771.023} C_VEL
LIN {X 0,Y 559.311,Z 123.157,A -85,B 0,C 180,E1 -2772.973,E2 -2772.973} C_VEL
LIN {X 0,Y 559.162,Z 137.013,A -85,B 0,C 180,E1 -2775.813,E2 -2775.813} C_VEL
LIN {X 0,Y 559.02,Z 152.073,A -85,B 0,C 180,E1 -2778.851,E2 -2778.851} C_VEL
LIN {X 0,Y 559.177,Z 153.527,A -85,B 0,C 180,E1 -2778.927,E2 -2778.927} C_VEL
LIN {X 0,Y 559.722,Z 158.879,A -85,B 0,C 180,E1 -2779.007,E2 -2779.007} C_VEL
LIN {X 0,Y 559.608,Z 228.527,A -85,B 0,C 180,E1 -2779.919,E2 -2779.919} C_VEL
LIN {X 0,Y 559.545,Z 238.987,A -85,B 0,C 180,E1 -2780.169,E2 -2780.169} C_VEL
LIN {X 0,Y 559.416,Z 250.617,A -85,B 0,C 180,E1 -2780.6,E2 -2780.6} C_VEL
LIN {X 0,Y 559.304,Z 261.091,A -85,B 0,C 180,E1 -2781.145,E2 -2781.145} C_VEL
LIN {X 0,Y 559.194,Z 270.485,A -85,B 0,C 180,E1 -2781.781,E2 -2781.781} C_VEL
LIN {X 0,Y 559.071,Z 279.897,A -85,B 0,C 180,E1 -2782.597,E2 -2782.597} C_VEL
LIN {X 0,Y 558.986,Z 288.006,A -85,B 0,C 180,E1 -2783.503,E2 -2783.503} C_VEL
LIN {X 0,Y 558.969,Z 293.315,A -85,B 0,C 180,E1 -2784.227,E2 -2784.227} C_VEL
LIN {X 0,Y 558.832,Z 297.75,A -85,B 0,C 180,E1 -2784.949,E2 -2784.949} C_VEL
LIN {X 0,Y 558.893,Z 301.443,A -85,B 0,C 180,E1 -2785.673,E2 -2785.673} C_VEL
LIN {X 0,Y 558.837,Z 305.643,A -85,B 0,C 180,E1 -2786.756,E2 -2786.756} C_VEL
LIN {X 0,Y 558.747,Z 308.582,A -85,B 0,C 180,E1 -2787.837,E2 -2787.837} C_VEL
LIN {X 0,Y 558.743,Z 309.871,A -85,B 0,C 180,E1 -2788.558,E2 -2788.558} C_VEL
LIN {X 0,Y 558.737,Z 310.688,A -85,B 0,C 180,E1 -2789.279,E2 -2789.279} C_VEL
LIN {X 0,Y 558.738,Z 310.996,A -85,B 0,C 180,E1 -2790,E2 -2790} C_VEL
LIN {X 0,Y 558.738,Z 310.728,A -85,B 0,C 180,E1 -2790.721,E2 -2790.721} C_VEL
LIN {X 0,Y 558.744,Z 309.991,A -85,B 0,C 180,E1 -2791.441,E2 -2791.441} C_VEL
LIN {X 0,Y 558.747,Z 308.785,A -85,B 0,C 180,E1 -2792.162,E2 -2792.162} C_VEL
LIN {X 0,Y 558.836,Z 305.932,A -85,B 0,C 180,E1 -2793.244,E2 -2793.244} C_VEL
LIN {X 0,Y 558.894,Z 301.822,A -85,B 0,C 180,E1 -2794.327,E2 -2794.327} C_VEL
LIN {X 0,Y 558.881,Z 296.244,A -85,B 0,C 180,E1 -2795.412,E2 -2795.412} C_VEL
LIN {X 0,Y 558.995,Z 290.132,A -85,B 0,C 180,E1 -2796.316,E2 -2796.316} C_VEL
LIN {X 0,Y 559.052,Z 284.349,A -85,B 0,C 180,E1 -2797.022,E2 -2797.022} C_VEL
LIN {X 0,Y 559.139,Z 275.996,A -85,B 0,C 180,E1 -2797.856,E2 -2797.856} C_VEL
LIN {X 0,Y 559.277,Z 266.733,A -85,B 0,C 180,E1 -2798.582,E2 -2798.582} C_VEL
LIN {X 0,Y 559.365,Z 256.221,A -85,B 0,C 180,E1 -2799.218,E2 -2799.218} C_VEL
LIN {X 0,Y 559.472,Z 246.13,A -85,B 0,C 180,E1 -2799.672,E2 -2799.672} C_VEL
LIN {X 0,Y 559.562,Z 236.45,A -85,B 0,C 180,E1 -2799.99,E2 -2799.99} C_VEL
LIN {X 0,Y 559.629,Z 227.169,A -85,B 0,C 180,E1 -2800.195,E2 -2800.195} C_VEL
LIN {X 0,Y 559.565,Z 156.243,A -85,B 0,C 180,E1 -2801.119,E2 -2801.119} C_VEL
LIN {X 0,Y 559.072,Z 152.825,A -85,B 0,C 180,E1 -2801.182,E2 -2801.182} C_VEL
LIN {X 0,Y 559.02,Z 151.67,A -85,B 0,C 180,E1 -2801.299,E2 -2801.299} C_VEL
LIN {X 0,Y 559.161,Z 137.477,A -85,B 0,C 180,E1 -2804.187,E2 -2804.187} C_VEL
LIN {X 0,Y 559.315,Z 122.464,A -85,B 0,C 180,E1 -2807.26,E2 -2807.26} C_VEL
LIN {X 0,Y 559.239,Z 113.741,A -85,B 0,C 180,E1 -2809.098,E2 -2809.098} C_VEL
LIN {X 0,Y 559.141,Z 113.648,A -85,B 0,C 180,E1 -2812.153,E2 -2812.153} C_VEL
LIN {X 0,Y 559.176,Z 113.639,A -85,B 0,C 180,E1 -2815.298,E2 -2815.298} C_VEL
LIN {X 0,Y 559.158,Z 113.642,A -85,B 0,C 180,E1 -2817.713,E2 -2817.713} C_VEL
LIN {X 0,Y 559.153,Z 113.65,A -85,B 0,C 180,E1 -2820.182,E2 -2820.182} C_VEL
LIN {X 0,Y 559.153,Z 113.644,A -85,B 0,C 180,E1 -2822.715,E2 -2822.715} C_VEL
LIN {X 0,Y 559.145,Z 113.643,A -85,B 0,C 180,E1 -2825.323,E2 -2825.323} C_VEL
LIN {X 0,Y 559.133,Z 113.653,A -85,B 0,C 180,E1 -2828.017,E2 -2828.017} C_VEL
LIN {X 0,Y 559.155,Z 113.642,A -85,B 0,C 180,E1 -2830.812,E2 -2830.812} C_VEL
LIN {X 0,Y 559.155,Z 113.651,A -85,B 0,C 180,E1 -2833.732,E2 -2833.732} C_VEL
LIN {X 0,Y 559.146,Z 113.643,A -85,B 0,C 180,E1 -2836.803,E2 -2836.803} C_VEL
LIN {X 0,Y 559.157,Z 113.645,A -85,B 0,C 180,E1 -2839.188,E2 -2839.188} C_VEL
LIN {X 0,Y 559.132,Z 113.646,A -85,B 0,C 180,E1 -2841.982,E2 -2841.982} C_VEL
LIN {X 0,Y 559.147,Z 113.645,A -85,B 0,C 180,E1 -2844.784,E2 -2844.784} C_VEL
LIN {X 0,Y 559.155,Z 113.649,A -85,B 0,C 180,E1 -2847.364,E2 -2847.364} C_VEL
LIN {X 0,Y 559.148,Z 113.642,A -85,B 0,C 180,E1 -2850.142,E2 -2850.142} C_VEL
LIN {X 0,Y 559.168,Z 113.648,A -85,B 0,C 180,E1 -2853.098,E2 -2853.098} C_VEL
LIN {X 0,Y 559.156,Z 113.643,A -85,B 0,C 180,E1 -2855.495,E2 -2855.495} C_VEL
LIN {X 0,Y 559.171,Z 113.646,A -85,B 0,C 180,E1 -2858.624,E2 -2858.624} C_VEL
LIN {X 0,Y 559.168,Z 113.646,A -85,B 0,C 180,E1 -2860.926,E2 -2860.926} C_VEL
LIN {X 0,Y 559.166,Z 113.641,A -85,B 0,C 180,E1 -2863.948,E2 -2863.948} C_VEL
LIN {X 0,Y 559.171,Z 113.644,A -85,B 0,C 180,E1 -2866.184,E2 -2866.184} C_VEL
LIN {X 0,Y 559.194,Z 113.637,A -85,B 0,C 180,E1 -2869.133,E2 -2869.133} C_VEL
LIN {X 0,Y 559.203,Z 113.641,A -85,B 0,C 180,E1 -2872.054,E2 -2872.054} C_VEL
LIN {X 0,Y 559.252,Z 113.63,A -85,B 0,C 180,E1 -2874.953,E2 -2874.953} C_VEL
LIN {X 0,Y 559.255,Z 113.635,A -85,B 0,C 180,E1 -2877.839,E2 -2877.839} C_VEL
LIN {X 0,Y 559.271,Z 113.628,A -85,B 0,C 180,E1 -2880.72,E2 -2880.72} C_VEL
LIN {X 0,Y 559.236,Z 113.631,A -85,B 0,C 180,E1 -2882.881,E2 -2882.881} C_VEL
LIN {X 0,Y 559.228,Z 113.642,A -85,B 0,C 180,E1 -2885.77,E2 -2885.77} C_VEL
LIN {X 0,Y 559.186,Z 113.638,A -85,B 0,C 180,E1 -2888.674,E2 -2888.674} C_VEL
LIN {X 0,Y 559.204,Z 113.644,A -85,B 0,C 180,E1 -2891.6,E2 -2891.6} C_VEL
LIN {X 0,Y 559.199,Z 113.636,A -85,B 0,C 180,E1 -2894.595,E2 -2894.595} C_VEL
LIN {X 0,Y 559.159,Z 113.646,A -85,B 0,C 180,E1 -2897.557,E2 -2897.557} C_VEL
LIN {X 0,Y 559.171,Z 113.641,A -85,B 0,C 180,E1 -2899.837,E2 -2899.837} C_VEL
LIN {X 0,Y 559.139,Z 113.643,A -85,B 0,C 180,E1 -2902.153,E2 -2902.153} C_VEL
LIN {X 0,Y 559.174,Z 113.644,A -85,B 0,C 180,E1 -2905.298,E2 -2905.298} C_VEL
LIN {X 0,Y 559.155,Z 113.642,A -85,B 0,C 180,E1 -2907.713,E2 -2907.713} C_VEL
LIN {X 0,Y 559.152,Z 113.643,A -85,B 0,C 180,E1 -2910.183,E2 -2910.183} C_VEL
LIN {X 0,Y 559.155,Z 113.651,A -85,B 0,C 180,E1 -2912.715,E2 -2912.715} C_VEL
LIN {X 0,Y 559.144,Z 113.644,A -85,B 0,C 180,E1 -2915.323,E2 -2915.323} C_VEL
LIN {X 0,Y 559.132,Z 113.647,A -85,B 0,C 180,E1 -2918.018,E2 -2918.018} C_VEL
LIN {X 0,Y 559.156,Z 113.645,A -85,B 0,C 180,E1 -2920.812,E2 -2920.812} C_VEL
LIN {X 0,Y 559.145,Z 113.643,A -85,B 0,C 180,E1 -2923.197,E2 -2923.197} C_VEL
LIN {X 0,Y 559.136,Z 113.652,A -85,B 0,C 180,E1 -2926.266,E2 -2926.266} C_VEL
LIN {X 0,Y 559.162,Z 113.641,A -85,B 0,C 180,E1 -2928.949,E2 -2928.949} C_VEL
LIN {X 0,Y 559.173,Z 113.64,A -85,B 0,C 180,E1 -2931.192,E2 -2931.192} C_VEL
LIN {X 0,Y 559.156,Z 113.649,A -85,B 0,C 180,E1 -2933.791,E2 -2933.791} C_VEL
LIN {X 0,Y 559.147,Z 113.644,A -85,B 0,C 180,E1 -2936.424,E2 -2936.424} C_VEL
LIN {X 0,Y 559.154,Z 113.642,A -85,B 0,C 180,E1 -2938.981,E2 -2938.981} C_VEL
LIN {X 0,Y 559.168,Z 113.65,A -85,B 0,C 180,E1 -2941.619,E2 -2941.619} C_VEL
LIN {X 0,Y 559.177,Z 113.643,A -85,B 0,C 180,E1 -2943.903,E2 -2943.903} C_VEL
LIN {X 0,Y 559.136,Z 113.635,A -85,B 0,C 180,E1 -2946.573,E2 -2946.573} C_VEL
LIN {X 0,Y 559.201,Z 113.801,A -85,B 0,C 180,E1 -2948.625,E2 -2948.625} C_VEL
LIN {X 0,Y 559.63,Z 117.952,A -85,B 0,C 180,E1 -2949.413,E2 -2949.413} C_VEL
LIN {X 0,Y 559.433,Z 134.832,A -85,B 0,C 180,E1 -2952.452,E2 -2952.452} C_VEL
LIN {X 0,Y 559.266,Z 149.803,A -85,B 0,C 180,E1 -2955.109,E2 -2955.109} C_VEL
LIN {X 0,Y 559.124,Z 167.493,A -85,B 0,C 180,E1 -2958.214,E2 -2958.214} C_VEL
LIN {X 0,Y 559.075,Z 171.196,A -85,B 0,C 180,E1 -2958.82,E2 -2958.82} C_VEL
LIN {X 0,Y 559.361,Z 173.771,A -85,B 0,C 180,E1 -2958.891,E2 -2958.891} C_VEL
LIN {X 0,Y 559.708,Z 179.529,A -85,B 0,C 180,E1 -2958.972,E2 -2958.972} C_VEL
LIN {X 0,Y 559.614,Z 247.13,A -85,B 0,C 180,E1 -2959.851,E2 -2959.851} C_VEL
LIN {X 0,Y 559.533,Z 256.401,A -85,B 0,C 180,E1 -2960.055,E2 -2960.055} C_VEL
LIN {X 0,Y 559.465,Z 264.879,A -85,B 0,C 180,E1 -2960.328,E2 -2960.328} C_VEL
LIN {X 0,Y 559.407,Z 273.391,A -85,B 0,C 180,E1 -2960.692,E2 -2960.692} C_VEL
LIN {X 0,Y 559.303,Z 281.724,A -85,B 0,C 180,E1 -2961.146,E2 -2961.146} C_VEL
LIN {X 0,Y 559.183,Z 289.761,A -85,B 0,C 180,E1 -2961.69,E2 -2961.69} C_VEL
LIN {X 0,Y 559.097,Z 298.434,A -85,B 0,C 180,E1 -2962.416,E2 -2962.416} C_VEL
LIN {X 0,Y 559.02,Z 306.826,A -85,B 0,C 180,E1 -2963.308,E2 -2963.308} C_VEL
LIN {X 0,Y 559.004,Z 312.438,A -85,B 0,C 180,E1 -2964.047,E2 -2964.047} C_VEL
LIN {X 0,Y 558.822,Z 317.99,A -85,B 0,C 180,E1 -2964.95,E2 -2964.95} C_VEL
LIN {X 0,Y 558.858,Z 323.15,A -85,B 0,C 180,E1 -2966.034,E2 -2966.034} C_VEL
LIN {X 0,Y 558.803,Z 326.938,A -85,B 0,C 180,E1 -2967.117,E2 -2967.117} C_VEL
LIN {X 0,Y 558.746,Z 328.681,A -85,B 0,C 180,E1 -2967.838,E2 -2967.838} C_VEL
LIN {X 0,Y 558.744,Z 329.93,A -85,B 0,C 180,E1 -2968.559,E2 -2968.559} C_VEL
LIN {X 0,Y 558.737,Z 330.707,A -85,B 0,C 180,E1 -2969.279,E2 -2969.279} C_VEL
LIN {X 0,Y 558.737,Z 331,A -85,B 0,C 180,E1 -2970,E2 -2970} C_VEL
LIN {X 0,Y 558.737,Z 330.706,A -85,B 0,C 180,E1 -2970.721,E2 -2970.721} C_VEL
LIN {X 0,Y 558.744,Z 329.929,A -85,B 0,C 180,E1 -2971.442,E2 -2971.442} C_VEL
LIN {X 0,Y 558.746,Z 328.679,A -85,B 0,C 180,E1 -2972.163,E2 -2972.163} C_VEL
LIN {X 0,Y 558.835,Z 325.786,A -85,B 0,C 180,E1 -2973.244,E2 -2973.244} C_VEL
LIN {X 0,Y 558.858,Z 323.148,A -85,B 0,C 180,E1 -2973.966,E2 -2973.966} C_VEL
LIN {X 0,Y 558.822,Z 317.985,A -85,B 0,C 180,E1 -2975.051,E2 -2975.051} C_VEL
LIN {X 0,Y 559.018,Z 311.181,A -85,B 0,C 180,E1 -2976.135,E2 -2976.135} C_VEL
LIN {X 0,Y 559.036,Z 303.74,A -85,B 0,C 180,E1 -2977.041,E2 -2977.041} C_VEL
LIN {X 0,Y 559.123,Z 296.395,A -85,B 0,C 180,E1 -2977.766,E2 -2977.766} C_VEL
LIN {X 0,Y 559.222,Z 288.531,A -85,B 0,C 180,E1 -2978.401,E2 -2978.401} C_VEL
LIN {X 0,Y 559.32,Z 280.218,A -85,B 0,C 180,E1 -2978.946,E2 -2978.946} C_VEL
LIN {X 0,Y 559.46,Z 269.603,A -85,B 0,C 180,E1 -2979.49,E2 -2979.49} C_VEL
LIN {X 0,Y 559.557,Z 258.056,A -85,B 0,C 180,E1 -2979.899,E2 -2979.899} C_VEL
LIN {X 0,Y 559.654,Z 248.41,A -85,B 0,C 180,E1 -2980.126,E2 -2980.126} C_VEL
LIN {X 0,Y 559.719,Z 189.087,A -85,B 0,C 180,E1 -2980.905,E2 -2980.905} C_VEL
LIN {X 0,Y 559.599,Z 175.668,A -85,B 0,C 180,E1 -2981.08,E2 -2981.08} C_VEL
LIN {X 0,Y 559.107,Z 171.473,A -85,B 0,C 180,E1 -2981.161,E2 -2981.161} C_VEL
LIN {X 0,Y 559.055,Z 170.177,A -85,B 0,C 180,E1 -2981.318,E2 -2981.318} C_VEL
LIN {X 0,Y 559.244,Z 153.805,A -85,B 0,C 180,E1 -2984.185,E2 -2984.185} C_VEL
LIN {X 0,Y 559.368,Z 137.686,A -85,B 0,C 180,E1 -2987.039,E2 -2987.039} C_VEL
LIN {X 0,Y 559.599,Z 122.173,A -85,B 0,C 180,E1 -2989.822,E2 -2989.822} C_VEL
LIN {X 0,Y 559.523,Z 115.838,A -85,B 0,C 180,E1 -2990.976,E2 -2990.976} C_VEL
LIN {X 0,Y 559.177,Z 113.67,A -85,B 0,C 180,E1 -2991.444,E2 -2991.444} C_VEL
LIN {X 0,Y 559.154,Z 113.641,A -85,B 0,C 180,E1 -2994.505,E2 -2994.505} C_VEL
LIN {X 0,Y 559.17,Z 113.642,A -85,B 0,C 180,E1 -2996.902,E2 -2996.902} C_VEL
LIN {X 0,Y 559.149,Z 113.645,A -85,B 0,C 180,E1 -2999.857,E2 -2999.857} C_VEL
LIN {X 0,Y 559.154,Z 113.644,A -85,B 0,C 180,E1 -3002.716,E2 -3002.716} C_VEL
LIN {X 0,Y 559.128,Z 113.645,A -85,B 0,C 180,E1 -3005.324,E2 -3005.324} C_VEL
LIN {X 0,Y 559.133,Z 113.654,A -85,B 0,C 180,E1 -3008.018,E2 -3008.018} C_VEL
LIN {X 0,Y 559.156,Z 113.641,A -85,B 0,C 180,E1 -3010.813,E2 -3010.813} C_VEL
LIN {X 0,Y 559.138,Z 113.652,A -85,B 0,C 180,E1 -3013.734,E2 -3013.734} C_VEL
LIN {X 0,Y 559.146,Z 113.643,A -85,B 0,C 180,E1 -3016.804,E2 -3016.804} C_VEL
LIN {X 0,Y 559.158,Z 113.644,A -85,B 0,C 180,E1 -3019.188,E2 -3019.188} C_VEL
LIN {X 0,Y 559.134,Z 113.647,A -85,B 0,C 180,E1 -3021.983,E2 -3021.983} C_VEL
LIN {X 0,Y 559.148,Z 113.644,A -85,B 0,C 180,E1 -3024.785,E2 -3024.785} C_VEL
LIN {X 0,Y 559.157,Z 113.65,A -85,B 0,C 180,E1 -3027.365,E2 -3027.365} C_VEL
LIN {X 0,Y 559.149,Z 113.642,A -85,B 0,C 180,E1 -3030.143,E2 -3030.143} C_VEL
LIN {X 0,Y 559.17,Z 113.649,A -85,B 0,C 180,E1 -3033.098,E2 -3033.098} C_VEL
LIN {X 0,Y 559.157,Z 113.644,A -85,B 0,C 180,E1 -3035.495,E2 -3035.495} C_VEL
LIN {X 0,Y 559.173,Z 113.645,A -85,B 0,C 180,E1 -3038.624,E2 -3038.624} C_VEL
LIN {X 0,Y 559.169,Z 113.647,A -85,B 0,C 180,E1 -3040.926,E2 -3040.926} C_VEL
LIN {X 0,Y 559.168,Z 113.641,A -85,B 0,C 180,E1 -3043.948,E2 -3043.948} C_VEL
LIN {X 0,Y 559.173,Z 113.643,A -85,B 0,C 180,E1 -3046.184,E2 -3046.184} C_VEL
LIN {X 0,Y 559.195,Z 113.638,A -85,B 0,C 180,E1 -3049.134,E2 -3049.134} C_VEL
LIN {X 0,Y 559.205,Z 113.64,A -85,B 0,C 180,E1 -3052.054,E2 -3052.054} C_VEL
LIN {X 0,Y 559.252,Z 113.63,A -85,B 0,C 180,E1 -3054.953,E2 -3054.953} C_VEL
LIN {X 0,Y 559.253,Z 113.634,A -85,B 0,C 180,E1 -3057.84,E2 -3057.84} C_VEL
LIN {X 0,Y 559.274,Z 113.628,A -85,B 0,C 180,E1 -3060.72,E2 -3060.72} C_VEL
LIN {X 0,Y 559.237,Z 113.631,A -85,B 0,C 180,E1 -3062.881,E2 -3062.881} C_VEL
LIN {X 0,Y 559.228,Z 113.641,A -85,B 0,C 180,E1 -3065.77,E2 -3065.77} C_VEL
LIN {X 0,Y 559.188,Z 113.637,A -85,B 0,C 180,E1 -3068.674,E2 -3068.674} C_VEL
LIN {X 0,Y 559.207,Z 113.644,A -85,B 0,C 180,E1 -3071.6,E2 -3071.6} C_VEL
LIN {X 0,Y 559.202,Z 113.636,A -85,B 0,C 180,E1 -3074.596,E2 -3074.596} C_VEL
LIN {X 0,Y 559.161,Z 113.648,A -85,B 0,C 180,E1 -3077.557,E2 -3077.557} C_VEL
LIN {X 0,Y 559.168,Z 113.642,A -85,B 0,C 180,E1 -3079.838,E2 -3079.838} C_VEL
LIN {X 0,Y 559.143,Z 113.643,A -85,B 0,C 180,E1 -3082.153,E2 -3082.153} C_VEL
LIN {X 0,Y 559.178,Z 113.645,A -85,B 0,C 180,E1 -3085.298,E2 -3085.298} C_VEL
LIN {X 0,Y 559.159,Z 113.642,A -85,B 0,C 180,E1 -3087.713,E2 -3087.713} C_VEL
LIN {X 0,Y 559.141,Z 113.646,A -85,B 0,C 180,E1 -3090.613,E2 -3090.613} C_VEL
LIN {X 0,Y 558.48,Z 113.733,A -85,B 0,C 180,E1 -3091.214,E2 -3091.214} C_VEL
LIN {X 0,Y 555.617,Z 114.088,A -85,B 0,C 180,E1 -3092.19,E2 -3092.19} C_VEL
LIN {X 0,Y 553.205,Z 114.39,A -85,B 0,C 180,E1 -3092.976,E2 -3092.976} C_VEL
LIN {X 0,Y 552.186,Z 114.511,A -85,B 0,C 180,E1 -3093.583,E2 -3093.583} C_VEL
LIN {X 0,Y 552.113,Z 114.519,A -85,B 0,C 180,E1 -3093.788,E2 -3093.788} C_VEL
LIN {X 0,Y 552.112,Z 114.528,A -85,B 0,C 180,E1 -3096.747,E2 -3096.747} C_VEL
LIN {X 0,Y 552.131,Z 114.516,A -85,B 0,C 180,E1 -3099.527,E2 -3099.527} C_VEL
LIN {X 0,Y 552.131,Z 114.525,A -85,B 0,C 180,E1 -3102.426,E2 -3102.426} C_VEL
LIN {X 0,Y 552.093,Z 114.522,A -85,B 0,C 180,E1 -3105.562,E2 -3105.562} C_VEL
LIN {X 0,Y 552.122,Z 114.522,A -85,B 0,C 180,E1 -3108.554,E2 -3108.554} C_VEL
LIN {X 0,Y 552.119,Z 114.519,A -85,B 0,C 180,E1 -3111.411,E2 -3111.411} C_VEL
LIN {X 0,Y 552.103,Z 114.527,A -85,B 0,C 180,E1 -3114.158,E2 -3114.158} C_VEL
LIN {X 0,Y 552.109,Z 114.519,A -85,B 0,C 180,E1 -3116.814,E2 -3116.814} C_VEL
LIN {X 0,Y 552.104,Z 114.523,A -85,B 0,C 180,E1 -3119.391,E2 -3119.391} C_VEL
LIN {X 0,Y 552.112,Z 114.526,A -85,B 0,C 180,E1 -3121.902,E2 -3121.902} C_VEL
LIN {X 0,Y 552.158,Z 114.513,A -85,B 0,C 180,E1 -3124.65,E2 -3124.65} C_VEL
LIN {X 0,Y 552.094,Z 114.531,A -85,B 0,C 180,E1 -3127.549,E2 -3127.549} C_VEL
LIN {X 0,Y 552.175,Z 114.516,A -85,B 0,C 180,E1 -3130.675,E2 -3130.675} C_VEL
LIN {X 0,Y 552.204,Z 114.707,A -85,B 0,C 180,E1 -3130.966,E2 -3130.966} C_VEL
LIN {X 0,Y 552.287,Z 124.27,A -85,B 0,C 180,E1 -3132.981,E2 -3132.981} C_VEL
LIN {X 0,Y 552.108,Z 138.876,A -85,B 0,C 180,E1 -3136.004,E2 -3136.004} C_VEL
LIN {X 0,Y 551.97,Z 152.248,A -85,B 0,C 180,E1 -3138.716,E2 -3138.716} C_VEL
LIN {X 0,Y 552.177,Z 153.869,A -85,B 0,C 180,E1 -3138.788,E2 -3138.788} C_VEL
LIN {X 0,Y 552.775,Z 160.17,A -85,B 0,C 180,E1 -3138.882,E2 -3138.882} C_VEL
LIN {X 0,Y 552.651,Z 227.388,A -85,B 0,C 180,E1 -3139.768,E2 -3139.768} C_VEL
LIN {X 0,Y 552.575,Z 236.635,A -85,B 0,C 180,E1 -3139.974,E2 -3139.974} C_VEL
LIN {X 0,Y 552.466,Z 246.297,A -85,B 0,C 180,E1 -3140.296,E2 -3140.296} C_VEL
LIN {X 0,Y 552.379,Z 256.375,A -85,B 0,C 180,E1 -3140.756,E2 -3140.756} C_VEL
LIN {X 0,Y 552.252,Z 266.834,A -85,B 0,C 180,E1 -3141.4,E2 -3141.4} C_VEL
LIN {X 0,Y 552.083,Z 274.999,A -85,B 0,C 180,E1 -3142.042,E2 -3142.042} C_VEL
LIN {X 0,Y 551.998,Z 281.731,A -85,B 0,C 180,E1 -3142.685,E2 -3142.685} C_VEL
LIN {X 0,Y 551.93,Z 288.105,A -85,B 0,C 180,E1 -3143.419,E2 -3143.419} C_VEL
LIN {X 0,Y 551.917,Z 293.402,A -85,B 0,C 180,E1 -3144.153,E2 -3144.153} C_VEL
LIN {X 0,Y 551.753,Z 297.827,A -85,B 0,C 180,E1 -3144.884,E2 -3144.884} C_VEL
LIN {X 0,Y 551.825,Z 301.508,A -85,B 0,C 180,E1 -3145.617,E2 -3145.617} C_VEL
LIN {X 0,Y 551.763,Z 305.696,A -85,B 0,C 180,E1 -3146.714,E2 -3146.714} C_VEL
LIN {X 0,Y 551.657,Z 308.626,A -85,B 0,C 180,E1 -3147.809,E2 -3147.809} C_VEL
LIN {X 0,Y 551.643,Z 309.91,A -85,B 0,C 180,E1 -3148.54,E2 -3148.54} C_VEL
LIN {X 0,Y 551.638,Z 310.725,A -85,B 0,C 180,E1 -3149.27,E2 -3149.27} C_VEL
LIN {X 0,Y 551.639,Z 311.033,A -85,B 0,C 180,E1 -3150,E2 -3150} C_VEL
LIN {X 0,Y 551.639,Z 310.764,A -85,B 0,C 180,E1 -3150.73,E2 -3150.73} C_VEL
LIN {X 0,Y 551.644,Z 310.029,A -85,B 0,C 180,E1 -3151.46,E2 -3151.46} C_VEL
LIN {X 0,Y 551.657,Z 308.826,A -85,B 0,C 180,E1 -3152.19,E2 -3152.19} C_VEL
LIN {X 0,Y 551.761,Z 305.981,A -85,B 0,C 180,E1 -3153.286,E2 -3153.286} C_VEL
LIN {X 0,Y 551.825,Z 301.882,A -85,B 0,C 180,E1 -3154.382,E2 -3154.382} C_VEL
LIN {X 0,Y 551.819,Z 296.317,A -85,B 0,C 180,E1 -3155.481,E2 -3155.481} C_VEL
LIN {X 0,Y 551.92,Z 289.958,A -85,B 0,C 180,E1 -3156.431,E2 -3156.431} C_VEL
LIN {X 0,Y 551.999,Z 284.268,A -85,B 0,C 180,E1 -3157.13,E2 -3157.13} C_VEL
LIN {X 0,Y 552.082,Z 277.019,A -85,B 0,C 180,E1 -3157.865,E2 -3157.865} C_VEL
LIN {X 0,Y 552.209,Z 269.271,A -85,B 0,C 180,E1 -3158.508,E2 -3158.508} C_VEL
LIN {X 0,Y 552.276,Z 261.103,A -85,B 0,C 180,E1 -3159.06,E2 -3159.06} C_VEL
LIN {X 0,Y 552.421,Z 252.59,A -85,B 0,C 180,E1 -3159.52,E2 -3159.52} C_VEL
LIN {X 0,Y 552.552,Z 242.606,A -85,B 0,C 180,E1 -3159.933,E2 -3159.933} C_VEL
LIN {X 0,Y 552.674,Z 231.157,A -85,B 0,C 180,E1 -3160.255,E2 -3160.255} C_VEL
LIN {X 0,Y 552.711,Z 212.421,A -85,B 0,C 180,E1 -3160.532,E2 -3160.532} C_VEL
LIN {X 0,Y 552.612,Z 156.794,A -85,B 0,C 180,E1 -3161.255,E2 -3161.255} C_VEL
LIN {X 0,Y 552.014,Z 152.667,A -85,B 0,C 180,E1 -3161.342,E2 -3161.342} C_VEL
LIN {X 0,Y 551.974,Z 151.558,A -85,B 0,C 180,E1 -3161.484,E2 -3161.484} C_VEL
LIN {X 0,Y 552.117,Z 137.687,A -85,B 0,C 180,E1 -3164.331,E2 -3164.331} C_VEL
LIN {X 0,Y 552.31,Z 122.98,A -85,B 0,C 180,E1 -3167.378,E2 -3167.378} C_VEL
LIN {X 0,Y 552.213,Z 114.606,A -85,B 0,C 180,E1 -3169.178,E2 -3169.178} C_VEL
LIN {X 0,Y 552.092,Z 114.53,A -85,B 0,C 180,E1 -3172.451,E2 -3172.451} C_VEL
LIN {X 0,Y 552.156,Z 114.513,A -85,B 0,C 180,E1 -3175.35,E2 -3175.35} C_VEL
LIN {X 0,Y 552.11,Z 114.525,A -85,B 0,C 180,E1 -3178.098,E2 -3178.098} C_VEL
LIN {X 0,Y 552.103,Z 114.524,A -85,B 0,C 180,E1 -3180.609,E2 -3180.609} C_VEL
LIN {X 0,Y 552.107,Z 114.519,A -85,B 0,C 180,E1 -3183.186,E2 -3183.186} C_VEL
LIN {X 0,Y 552.101,Z 114.526,A -85,B 0,C 180,E1 -3185.842,E2 -3185.842} C_VEL
LIN {X 0,Y 552.121,Z 114.518,A -85,B 0,C 180,E1 -3189.061,E2 -3189.061} C_VEL
LIN {X 0,Y 552.12,Z 114.521,A -85,B 0,C 180,E1 -3191.446,E2 -3191.446} C_VEL
LIN {X 0,Y 552.09,Z 114.522,A -85,B 0,C 180,E1 -3194.531,E2 -3194.531} C_VEL
LIN {X 0,Y 552.13,Z 114.526,A -85,B 0,C 180,E1 -3197.584,E2 -3197.584} C_VEL
LIN {X 0,Y 552.129,Z 114.517,A -85,B 0,C 180,E1 -3200.473,E2 -3200.473} C_VEL
LIN {X 0,Y 552.111,Z 114.527,A -85,B 0,C 180,E1 -3203.316,E2 -3203.316} C_VEL
LIN {X 0,Y 552.128,Z 114.518,A -85,B 0,C 180,E1 -3205.939,E2 -3205.939} C_VEL
LIN {X 0,Y 552.118,Z 114.519,A -85,B 0,C 180,E1 -3208.54,E2 -3208.54} C_VEL
LIN {X 0,Y 552.124,Z 114.521,A -85,B 0,C 180,E1 -3211.438,E2 -3211.438} C_VEL
LIN {X 0,Y 552.129,Z 114.518,A -85,B 0,C 180,E1 -3214.356,E2 -3214.356} C_VEL
LIN {X 0,Y 552.098,Z 114.528,A -85,B 0,C 180,E1 -3216.758,E2 -3216.758} C_VEL
LIN {X 0,Y 552.12,Z 114.522,A -85,B 0,C 180,E1 -3219.12,E2 -3219.12} C_VEL
LIN {X 0,Y 552.125,Z 114.518,A -85,B 0,C 180,E1 -3221.444,E2 -3221.444} C_VEL
LIN {X 0,Y 552.116,Z 114.519,A -85,B 0,C 180,E1 -3223.737,E2 -3223.737} C_VEL
LIN {X 0,Y 552.135,Z 114.518,A -85,B 0,C 180,E1 -3226.004,E2 -3226.004} C_VEL
LIN {X 0,Y 552.162,Z 114.514,A -85,B 0,C 180,E1 -3228.993,E2 -3228.993} C_VEL
LIN {X 0,Y 552.157,Z 114.518,A -85,B 0,C 180,E1 -3231.951,E2 -3231.951} C_VEL
LIN {X 0,Y 552.227,Z 114.505,A -85,B 0,C 180,E1 -3234.889,E2 -3234.889} C_VEL
LIN {X 0,Y 552.226,Z 114.51,A -85,B 0,C 180,E1 -3237.812,E2 -3237.812} C_VEL
LIN {X 0,Y 552.241,Z 114.503,A -85,B 0,C 180,E1 -3240.729,E2 -3240.729} C_VEL
LIN {X 0,Y 552.203,Z 114.508,A -85,B 0,C 180,E1 -3242.918,E2 -3242.918} C_VEL
LIN {X 0,Y 552.198,Z 114.516,A -85,B 0,C 180,E1 -3245.844,E2 -3245.844} C_VEL
LIN {X 0,Y 552.157,Z 114.513,A -85,B 0,C 180,E1 -3248.786,E2 -3248.786} C_VEL
LIN {X 0,Y 552.162,Z 114.518,A -85,B 0,C 180,E1 -3251.75,E2 -3251.75} C_VEL
LIN {X 0,Y 552.135,Z 114.517,A -85,B 0,C 180,E1 -3254.748,E2 -3254.748} C_VEL
LIN {X 0,Y 552.11,Z 114.522,A -85,B 0,C 180,E1 -3257.788,E2 -3257.788} C_VEL
LIN {X 0,Y 552.13,Z 114.517,A -85,B 0,C 180,E1 -3260.101,E2 -3260.101} C_VEL
LIN {X 0,Y 552.09,Z 114.523,A -85,B 0,C 180,E1 -3262.451,E2 -3262.451} C_VEL
LIN {X 0,Y 552.154,Z 114.518,A -85,B 0,C 180,E1 -3265.35,E2 -3265.35} C_VEL
LIN {X 0,Y 552.108,Z 114.52,A -85,B 0,C 180,E1 -3268.098,E2 -3268.098} C_VEL
LIN {X 0,Y 552.101,Z 114.527,A -85,B 0,C 180,E1 -3270.609,E2 -3270.609} C_VEL
LIN {X 0,Y 552.114,Z 114.521,A -85,B 0,C 180,E1 -3273.186,E2 -3273.186} C_VEL
LIN {X 0,Y 552.102,Z 114.521,A -85,B 0,C 180,E1 -3275.842,E2 -3275.842} C_VEL
LIN {X 0,Y 552.12,Z 114.52,A -85,B 0,C 180,E1 -3279.061,E2 -3279.061} C_VEL
LIN {X 0,Y 552.128,Z 114.517,A -85,B 0,C 180,E1 -3281.445,E2 -3281.445} C_VEL
LIN {X 0,Y 552.091,Z 114.527,A -85,B 0,C 180,E1 -3284.532,E2 -3284.532} C_VEL
LIN {X 0,Y 552.129,Z 114.519,A -85,B 0,C 180,E1 -3287.585,E2 -3287.585} C_VEL
LIN {X 0,Y 552.128,Z 114.52,A -85,B 0,C 180,E1 -3290.473,E2 -3290.473} C_VEL
LIN {X 0,Y 552.11,Z 114.521,A -85,B 0,C 180,E1 -3293.317,E2 -3293.317} C_VEL
LIN {X 0,Y 552.121,Z 114.525,A -85,B 0,C 180,E1 -3295.939,E2 -3295.939} C_VEL
LIN {X 0,Y 552.118,Z 114.518,A -85,B 0,C 180,E1 -3298.541,E2 -3298.541} C_VEL
LIN {X 0,Y 552.124,Z 114.524,A -85,B 0,C 180,E1 -3301.438,E2 -3301.438} C_VEL
LIN {X 0,Y 552.128,Z 114.517,A -85,B 0,C 180,E1 -3304.356,E2 -3304.356} C_VEL
LIN {X 0,Y 552.094,Z 114.512,A -85,B 0,C 180,E1 -3306.758,E2 -3306.758} C_VEL
LIN {X 0,Y 552.181,Z 114.727,A -85,B 0,C 180,E1 -3308.536,E2 -3308.536} C_VEL
LIN {X 0,Y 552.628,Z 119.95,A -85,B 0,C 180,E1 -3309.53,E2 -3309.53} C_VEL
LIN {X 0,Y 552.398,Z 136.085,A -85,B 0,C 180,E1 -3312.47,E2 -3312.47} C_VEL
LIN {X 0,Y 552.201,Z 151.833,A -85,B 0,C 180,E1 -3315.3,E2 -3315.3} C_VEL
LIN {X 0,Y 552.048,Z 168.417,A -85,B 0,C 180,E1 -3318.247,E2 -3318.247} C_VEL
LIN {X 0,Y 552.023,Z 171.067,A -85,B 0,C 180,E1 -3318.676,E2 -3318.676} C_VEL
LIN {X 0,Y 552.406,Z 174.478,A -85,B 0,C 180,E1 -3318.761,E2 -3318.761} C_VEL
LIN {X 0,Y 552.77,Z 182.198,A -85,B 0,C 180,E1 -3318.868,E2 -3318.868} C_VEL
LIN {X 0,Y 552.649,Z 247.002,A -85,B 0,C 180,E1 -3319.722,E2 -3319.722} C_VEL
LIN {X 0,Y 552.551,Z 256.273,A -85,B 0,C 180,E1 -3319.928,E2 -3319.928} C_VEL
LIN {X 0,Y 552.48,Z 264.751,A -85,B 0,C 180,E1 -3320.204,E2 -3320.204} C_VEL
LIN {X 0,Y 552.397,Z 273.264,A -85,B 0,C 180,E1 -3320.572,E2 -3320.572} C_VEL
LIN {X 0,Y 552.266,Z 281.608,A -85,B 0,C 180,E1 -3321.032,E2 -3321.032} C_VEL
LIN {X 0,Y 552.142,Z 289.658,A -85,B 0,C 180,E1 -3321.583,E2 -3321.583} C_VEL
LIN {X 0,Y 552.031,Z 298.346,A -85,B 0,C 180,E1 -3322.318,E2 -3322.318} C_VEL
LIN {X 0,Y 551.953,Z 307.366,A -85,B 0,C 180,E1 -3323.3,E2 -3323.3} C_VEL
LIN {X 0,Y 551.895,Z 313.559,A -85,B 0,C 180,E1 -3324.153,E2 -3324.153} C_VEL
LIN {X 0,Y 551.743,Z 317.948,A -85,B 0,C 180,E1 -3324.885,E2 -3324.885} C_VEL
LIN {X 0,Y 551.778,Z 323.125,A -85,B 0,C 180,E1 -3325.983,E2 -3325.983} C_VEL
LIN {X 0,Y 551.729,Z 326.924,A -85,B 0,C 180,E1 -3327.08,E2 -3327.08} C_VEL
LIN {X 0,Y 551.657,Z 328.67,A -85,B 0,C 180,E1 -3327.81,E2 -3327.81} C_VEL
LIN {X 0,Y 551.643,Z 329.922,A -85,B 0,C 180,E1 -3328.54,E2 -3328.54} C_VEL
LIN {X 0,Y 551.638,Z 330.702,A -85,B 0,C 180,E1 -3329.27,E2 -3329.27} C_VEL
LIN {X 0,Y 551.637,Z 330.997,A -85,B 0,C 180,E1 -3330,E2 -3330} C_VEL
LIN {X 0,Y 551.638,Z 330.701,A -85,B 0,C 180,E1 -3330.73,E2 -3330.73} C_VEL
LIN {X 0,Y 551.643,Z 329.921,A -85,B 0,C 180,E1 -3331.46,E2 -3331.46} C_VEL
LIN {X 0,Y 551.657,Z 328.668,A -85,B 0,C 180,E1 -3332.191,E2 -3332.191} C_VEL
LIN {X 0,Y 551.761,Z 325.768,A -85,B 0,C 180,E1 -3333.286,E2 -3333.286} C_VEL
LIN {X 0,Y 551.778,Z 323.123,A -85,B 0,C 180,E1 -3334.017,E2 -3334.017} C_VEL
LIN {X 0,Y 551.743,Z 317.943,A -85,B 0,C 180,E1 -3335.116,E2 -3335.116} C_VEL
LIN {X 0,Y 551.936,Z 311.34,A -85,B 0,C 180,E1 -3336.184,E2 -3336.184} C_VEL
LIN {X 0,Y 551.969,Z 303.664,A -85,B 0,C 180,E1 -3337.131,E2 -3337.131} C_VEL
LIN {X 0,Y 552.079,Z 296.304,A -85,B 0,C 180,E1 -3337.866,E2 -3337.866} C_VEL
LIN {X 0,Y 552.195,Z 288.426,A -85,B 0,C 180,E1 -3338.509,E2 -3338.509} C_VEL
LIN {X 0,Y 552.298,Z 280.101,A -85,B 0,C 180,E1 -3339.06,E2 -3339.06} C_VEL
LIN {X 0,Y 552.46,Z 269.475,A -85,B 0,C 180,E1 -3339.612,E2 -3339.612} C_VEL
LIN {X 0,Y 552.563,Z 257.928,A -85,B 0,C 180,E1 -3340.026,E2 -3340.026} C_VEL
LIN {X 0,Y 552.638,Z 249.578,A -85,B 0,C 180,E1 -3340.233,E2 -3340.233} C_VEL
LIN {X 0,Y 552.707,Z 226.792,A -85,B 0,C 180,E1 -3340.555,E2 -3340.555} C_VEL
LIN {X 0,Y 552.588,Z 175.86,A -85,B 0,C 180,E1 -3341.218,E2 -3341.218} C_VEL
LIN {X 0,Y 552.027,Z 171.332,A -85,B 0,C 180,E1 -3341.306,E2 -3341.306} C_VEL
LIN {X 0,Y 552.016,Z 169.878,A -85,B 0,C 180,E1 -3341.495,E2 -3341.495} C_VEL
LIN {X 0,Y 552.188,Z 153.806,A -85,B 0,C 180,E1 -3344.347,E2 -3344.347} C_VEL
LIN {X 0,Y 552.341,Z 138.927,A -85,B 0,C 180,E1 -3347.017,E2 -3347.017} C_VEL
LIN {X 0,Y 552.566,Z 123.896,A -85,B 0,C 180,E1 -3349.747,E2 -3349.747} C_VEL
LIN {X 0,Y 552.52,Z 116.781,A -85,B 0,C 180,E1 -3351.06,E2 -3351.06} C_VEL
LIN {X 0,Y 552.129,Z 114.547,A -85,B 0,C 180,E1 -3351.549,E2 -3351.549} C_VEL
LIN {X 0,Y 552.1,Z 114.51,A -85,B 0,C 180,E1 -3354.038,E2 -3354.038} C_VEL
LIN {X 0,Y 552.12,Z 114.528,A -85,B 0,C 180,E1 -3356.457,E2 -3356.457} C_VEL
LIN {X 0,Y 552.111,Z 114.521,A -85,B 0,C 180,E1 -3358.928,E2 -3358.928} C_VEL
LIN {X 0,Y 552.112,Z 114.519,A -85,B 0,C 180,E1 -3361.476,E2 -3361.476} C_VEL
LIN {X 0,Y 552.133,Z 114.526,A -85,B 0,C 180,E1 -3364.17,E2 -3364.17} C_VEL
LIN {X 0,Y 552.106,Z 114.521,A -85,B 0,C 180,E1 -3366.747,E2 -3366.747} C_VEL
LIN {X 0,Y 552.13,Z 114.52,A -85,B 0,C 180,E1 -3369.527,E2 -3369.527} C_VEL
LIN {X 0,Y 552.13,Z 114.518,A -85,B 0,C 180,E1 -3372.426,E2 -3372.426} C_VEL
LIN {X 0,Y 552.092,Z 114.528,A -85,B 0,C 180,E1 -3375.562,E2 -3375.562} C_VEL
LIN {X 0,Y 552.131,Z 114.517,A -85,B 0,C 180,E1 -3378.555,E2 -3378.555} C_VEL
LIN {X 0,Y 552.118,Z 114.526,A -85,B 0,C 180,E1 -3381.411,E2 -3381.411} C_VEL
LIN {X 0,Y 552.104,Z 114.521,A -85,B 0,C 180,E1 -3384.158,E2 -3384.158} C_VEL
LIN {X 0,Y 552.116,Z 114.521,A -85,B 0,C 180,E1 -3386.814,E2 -3386.814} C_VEL
LIN {X 0,Y 552.103,Z 114.527,A -85,B 0,C 180,E1 -3389.391,E2 -3389.391} C_VEL
LIN {X 0,Y 552.111,Z 114.52,A -85,B 0,C 180,E1 -3391.902,E2 -3391.902} C_VEL
LIN {X 0,Y 552.156,Z 114.517,A -85,B 0,C 180,E1 -3394.65,E2 -3394.65} C_VEL
LIN {X 0,Y 552.093,Z 114.523,A -85,B 0,C 180,E1 -3397.549,E2 -3397.549} C_VEL
LIN {X 0,Y 552.15,Z 114.517,A -85,B 0,C 180,E1 -3400.374,E2 -3400.374} C_VEL
LIN {X 0,Y 552.157,Z 114.518,A -85,B 0,C 180,E1 -3402.977,E2 -3402.977} C_VEL
LIN {X 0,Y 552.137,Z 114.517,A -85,B 0,C 180,E1 -3406.005,E2 -3406.005} C_VEL
LIN {X 0,Y 552.163,Z 114.515,A -85,B 0,C 180,E1 -3408.993,E2 -3408.993} C_VEL
LIN {X 0,Y 552.159,Z 114.516,A -85,B 0,C 180,E1 -3411.952,E2 -3411.952} C_VEL
LIN {X 0,Y 552.227,Z 114.506,A -85,B 0,C 180,E1 -3414.889,E2 -3414.889} C_VEL
LIN {X 0,Y 552.225,Z 114.509,A -85,B 0,C 180,E1 -3417.812,E2 -3417.812} C_VEL
LIN {X 0,Y 552.244,Z 114.503,A -85,B 0,C 180,E1 -3420.729,E2 -3420.729} C_VEL
LIN {X 0,Y 552.204,Z 114.507,A -85,B 0,C 180,E1 -3422.918,E2 -3422.918} C_VEL
LIN {X 0,Y 552.199,Z 114.518,A -85,B 0,C 180,E1 -3425.844,E2 -3425.844} C_VEL
LIN {X 0,Y 552.159,Z 114.513,A -85,B 0,C 180,E1 -3428.786,E2 -3428.786} C_VEL
LIN {X 0,Y 552.165,Z 114.52,A -85,B 0,C 180,E1 -3431.751,E2 -3431.751} C_VEL
LIN {X 0,Y 552.139,Z 114.516,A -85,B 0,C 180,E1 -3434.748,E2 -3434.748} C_VEL
LIN {X 0,Y 552.111,Z 114.523,A -85,B 0,C 180,E1 -3437.789,E2 -3437.789} C_VEL
LIN {X 0,Y 552.129,Z 114.517,A -85,B 0,C 180,E1 -3440.101,E2 -3440.101} C_VEL
LIN {X 0,Y 552.094,Z 114.522,A -85,B 0,C 180,E1 -3442.451,E2 -3442.451} C_VEL
LIN {X 0,Y 552.157,Z 114.519,A -85,B 0,C 180,E1 -3445.35,E2 -3445.35} C_VEL
LIN {X 0,Y 552.111,Z 114.519,A -85,B 0,C 180,E1 -3448.098,E2 -3448.098} C_VEL
LIN {X 0,Y 552.105,Z 114.524,A -85,B 0,C 180,E1 -3450.609,E2 -3450.609} C_VEL
LIN {X 0,Y 552.117,Z 114.522,A -85,B 0,C 180,E1 -3453.186,E2 -3453.186} C_VEL
LIN {X 0,Y 552.113,Z 114.519,A -85,B 0,C 180,E1 -3453.788,E2 -3453.788} C_VEL
LIN {X 0,Y 551.48,Z 114.602,A -85,B 0,C 180,E1 -3454.397,E2 -3454.397} C_VEL
LIN {X 0,Y 548.66,Z 114.957,A -85,B 0,C 180,E1 -3455.385,E2 -3455.385} C_VEL
LIN {X 0,Y 546.239,Z 115.261,A -85,B 0,C 180,E1 -3456.18,E2 -3456.18} C_VEL
LIN {X 0,Y 545.169,Z 115.391,A -85,B 0,C 180,E1 -3456.794,E2 -3456.794} C_VEL
LIN {X 0,Y 545.066,Z 115.401,A -85,B 0,C 180,E1 -3457.002,E2 -3457.002} C_VEL
LIN {X 0,Y 545.067,Z 115.4,A -85,B 0,C 180,E1 -3460.143,E2 -3460.143} C_VEL
LIN {X 0,Y 545.08,Z 115.396,A -85,B 0,C 180,E1 -3463.107,E2 -3463.107} C_VEL
LIN {X 0,Y 545.05,Z 115.406,A -85,B 0,C 180,E1 -3466.226,E2 -3466.226} C_VEL
LIN {X 0,Y 545.083,Z 115.396,A -85,B 0,C 180,E1 -3468.885,E2 -3468.885} C_VEL
LIN {X 0,Y 545.082,Z 115.396,A -85,B 0,C 180,E1 -3470.818,E2 -3470.818} C_VEL
LIN {X 0,Y 545.051,Z 115.401,A -85,B 0,C 180,E1 -3473.62,E2 -3473.62} C_VEL
LIN {X 0,Y 545.062,Z 115.401,A -85,B 0,C 180,E1 -3476.328,E2 -3476.328} C_VEL
LIN {X 0,Y 545.068,Z 115.396,A -85,B 0,C 180,E1 -3478.952,E2 -3478.952} C_VEL
LIN {X 0,Y 545.103,Z 115.397,A -85,B 0,C 180,E1 -3481.508,E2 -3481.508} C_VEL
LIN {X 0,Y 545.097,Z 115.393,A -85,B 0,C 180,E1 -3484.491,E2 -3484.491} C_VEL
LIN {X 0,Y 545.038,Z 115.406,A -85,B 0,C 180,E1 -3487.242,E2 -3487.242} C_VEL
LIN {X 0,Y 545.121,Z 115.394,A -85,B 0,C 180,E1 -3490.415,E2 -3490.415} C_VEL
LIN {X 0,Y 545.173,Z 115.612,A -85,B 0,C 180,E1 -3490.906,E2 -3490.906} C_VEL
LIN {X 0,Y 545.285,Z 124.279,A -85,B 0,C 180,E1 -3492.756,E2 -3492.756} C_VEL
LIN {X 0,Y 545.084,Z 138.913,A -85,B 0,C 180,E1 -3495.82,E2 -3495.82} C_VEL
LIN {X 0,Y 544.931,Z 152.411,A -85,B 0,C 180,E1 -3498.573,E2 -3498.573} C_VEL
LIN {X 0,Y 545.229,Z 154.567,A -85,B 0,C 180,E1 -3498.65,E2 -3498.65} C_VEL
LIN {X 0,Y 545.824,Z 160.984,A -85,B 0,C 180,E1 -3498.747,E2 -3498.747} C_VEL
LIN {X 0,Y 545.678,Z 227.547,A -85,B 0,C 180,E1 -3499.635,E2 -3499.635} C_VEL
LIN {X 0,Y 545.595,Z 236.78,A -85,B 0,C 180,E1 -3499.845,E2 -3499.845} C_VEL
LIN {X 0,Y 545.488,Z 246.436,A -85,B 0,C 180,E1 -3500.171,E2 -3500.171} C_VEL
LIN {X 0,Y 545.376,Z 256.513,A -85,B 0,C 180,E1 -3500.637,E2 -3500.637} C_VEL
LIN {X 0,Y 545.243,Z 266.971,A -85,B 0,C 180,E1 -3501.289,E2 -3501.289} C_VEL
LIN {X 0,Y 545.05,Z 275.134,A -85,B 0,C 180,E1 -3501.939,E2 -3501.939} C_VEL
LIN {X 0,Y 544.946,Z 281.866,A -85,B 0,C 180,E1 -3502.59,E2 -3502.59} C_VEL
LIN {X 0,Y 544.881,Z 288.238,A -85,B 0,C 180,E1 -3503.334,E2 -3503.334} C_VEL
LIN {X 0,Y 544.868,Z 293.533,A -85,B 0,C 180,E1 -3504.077,E2 -3504.077} C_VEL
LIN {X 0,Y 544.678,Z 297.957,A -85,B 0,C 180,E1 -3504.818,E2 -3504.818} C_VEL
LIN {X 0,Y 544.757,Z 301.638,A -85,B 0,C 180,E1 -3505.56,E2 -3505.56} C_VEL
LIN {X 0,Y 544.69,Z 305.826,A -85,B 0,C 180,E1 -3506.671,E2 -3506.671} C_VEL
LIN {X 0,Y 544.572,Z 308.755,A -85,B 0,C 180,E1 -3507.781,E2 -3507.781} C_VEL
LIN {X 0,Y 544.545,Z 310.038,A -85,B 0,C 180,E1 -3508.521,E2 -3508.521} C_VEL
LIN {X 0,Y 544.539,Z 310.853,A -85,B 0,C 180,E1 -3509.26,E2 -3509.26} C_VEL
LIN {X 0,Y 544.54,Z 311.161,A -85,B 0,C 180,E1 -3510,E2 -3510} C_VEL
LIN {X 0,Y 544.54,Z 310.892,A -85,B 0,C 180,E1 -3510.739,E2 -3510.739} C_VEL
LIN {X 0,Y 544.546,Z 310.156,A -85,B 0,C 180,E1 -3511.479,E2 -3511.479} C_VEL
LIN {X 0,Y 544.572,Z 308.953,A -85,B 0,C 180,E1 -3512.219,E2 -3512.219} C_VEL
LIN {X 0,Y 544.688,Z 306.107,A -85,B 0,C 180,E1 -3513.328,E2 -3513.328} C_VEL
LIN {X 0,Y 544.7,Z 303.522,A -85,B 0,C 180,E1 -3514.069,E2 -3514.069} C_VEL
LIN {X 0,Y 544.667,Z 298.423,A -85,B 0,C 180,E1 -3515.182,E2 -3515.182} C_VEL
LIN {X 0,Y 544.904,Z 292.482,A -85,B 0,C 180,E1 -3516.18,E2 -3516.18} C_VEL
LIN {X 0,Y 544.946,Z 284.388,A -85,B 0,C 180,E1 -3517.223,E2 -3517.223} C_VEL
LIN {X 0,Y 545.04,Z 277.138,A -85,B 0,C 180,E1 -3517.968,E2 -3517.968} C_VEL
LIN {X 0,Y 545.197,Z 269.391,A -85,B 0,C 180,E1 -3518.618,E2 -3518.618} C_VEL
LIN {X 0,Y 545.27,Z 261.224,A -85,B 0,C 180,E1 -3519.178,E2 -3519.178} C_VEL
LIN {X 0,Y 545.495,Z 250.832,A -85,B 0,C 180,E1 -3519.735,E2 -3519.735} C_VEL
LIN {X 0,Y 545.589,Z 239.151,A -85,B 0,C 180,E1 -3520.178,E2 -3520.178} C_VEL
LIN {X 0,Y 545.72,Z 228.653,A -85,B 0,C 180,E1 -3520.434,E2 -3520.434} C_VEL
LIN {X 0,Y 545.743,Z 158.011,A -85,B 0,C 180,E1 -3521.384,E2 -3521.384} C_VEL
LIN {X 0,Y 544.985,Z 152.9,A -85,B 0,C 180,E1 -3521.482,E2 -3521.482} C_VEL
LIN {X 0,Y 544.937,Z 151.656,A -85,B 0,C 180,E1 -3521.632,E2 -3521.632} C_VEL
LIN {X 0,Y 545.083,Z 136.575,A -85,B 0,C 180,E1 -3524.758,E2 -3524.758} C_VEL
LIN {X 0,Y 545.308,Z 121.044,A -85,B 0,C 180,E1 -3528.018,E2 -3528.018} C_VEL
LIN {X 0,Y 545.171,Z 115.489,A -85,B 0,C 180,E1 -3529.24,E2 -3529.24} C_VEL
LIN {X 0,Y 545.048,Z 115.403,A -85,B 0,C 180,E1 -3531.958,E2 -3531.958} C_VEL
LIN {X 0,Y 545.049,Z 115.407,A -85,B 0,C 180,E1 -3534.369,E2 -3534.369} C_VEL
LIN {X 0,Y 545.088,Z 115.394,A -85,B 0,C 180,E1 -3537.172,E2 -3537.172} C_VEL
LIN {X 0,Y 545.065,Z 115.397,A -85,B 0,C 180,E1 -3539.338,E2 -3539.338} C_VEL
LIN {X 0,Y 545.055,Z 115.403,A -85,B 0,C 180,E1 -3541.915,E2 -3541.915} C_VEL
LIN {X 0,Y 545.075,Z 115.398,A -85,B 0,C 180,E1 -3544.563,E2 -3544.563} C_VEL
LIN {X 0,Y 545.038,Z 115.401,A -85,B 0,C 180,E1 -3547.304,E2 -3547.304} C_VEL
LIN {X 0,Y 545.066,Z 115.402,A -85,B 0,C 180,E1 -3550.142,E2 -3550.142} C_VEL
LIN {X 0,Y 545.078,Z 115.396,A -85,B 0,C 180,E1 -3553.106,E2 -3553.106} C_VEL
LIN {X 0,Y 545.049,Z 115.4,A -85,B 0,C 180,E1 -3556.226,E2 -3556.226} C_VEL
LIN {X 0,Y 545.085,Z 115.395,A -85,B 0,C 180,E1 -3558.886,E2 -3558.886} C_VEL
LIN {X 0,Y 545.051,Z 115.403,A -85,B 0,C 180,E1 -3561.762,E2 -3561.762} C_VEL
LIN {X 0,Y 545.053,Z 115.399,A -85,B 0,C 180,E1 -3564.533,E2 -3564.533} C_VEL
LIN {X 0,Y 545.068,Z 115.406,A -85,B 0,C 180,E1 -3567.211,E2 -3567.211} C_VEL
LIN {X 0,Y 545.063,Z 115.398,A -85,B 0,C 180,E1 -3569.81,E2 -3569.81} C_VEL
LIN {X 0,Y 545.08,Z 115.396,A -85,B 0,C 180,E1 -3572.344,E2 -3572.344} C_VEL
LIN {X 0,Y 545.116,Z 115.398,A -85,B 0,C 180,E1 -3574.82,E2 -3574.82} C_VEL
LIN {X 0,Y 545.037,Z 115.404,A -85,B 0,C 180,E1 -3577.242,E2 -3577.242} C_VEL
LIN {X 0,Y 545.12,Z 115.395,A -85,B 0,C 180,E1 -3580.415,E2 -3580.415} C_VEL
LIN {X 0,Y 545.072,Z 115.396,A -85,B 0,C 180,E1 -3583.521,E2 -3583.521} C_VEL
LIN {X 0,Y 545.094,Z 115.394,A -85,B 0,C 180,E1 -3585.82,E2 -3585.82} C_VEL
LIN {X 0,Y 545.117,Z 115.393,A -85,B 0,C 180,E1 -3588.849,E2 -3588.849} C_VEL
LIN {X 0,Y 545.128,Z 115.392,A -85,B 0,C 180,E1 -3591.847,E2 -3591.847} C_VEL
LIN {X 0,Y 545.203,Z 115.381,A -85,B 0,C 180,E1 -3594.823,E2 -3594.823} C_VEL
LIN {X 0,Y 545.197,Z 115.385,A -85,B 0,C 180,E1 -3597.784,E2 -3597.784} C_VEL
LIN {X 0,Y 545.211,Z 115.379,A -85,B 0,C 180,E1 -3600.739,E2 -3600.739} C_VEL
LIN {X 0,Y 545.17,Z 115.384,A -85,B 0,C 180,E1 -3602.956,E2 -3602.956} C_VEL
LIN {X 0,Y 545.17,Z 115.39,A -85,B 0,C 180,E1 -3605.919,E2 -3605.919} C_VEL
LIN {X 0,Y 545.116,Z 115.391,A -85,B 0,C 180,E1 -3608.9,E2 -3608.9} C_VEL
LIN {X 0,Y 545.134,Z 115.392,A -85,B 0,C 180,E1 -3611.904,E2 -3611.904} C_VEL
LIN {X 0,Y 545.084,Z 115.397,A -85,B 0,C 180,E1 -3614.944,E2 -3614.944} C_VEL
LIN {X 0,Y 545.078,Z 115.396,A -85,B 0,C 180,E1 -3618.026,E2 -3618.026} C_VEL
LIN {X 0,Y 545.094,Z 115.393,A -85,B 0,C 180,E1 -3620.372,E2 -3620.372} C_VEL
LIN {X 0,Y 545.077,Z 115.398,A -85,B 0,C 180,E1 -3623.559,E2 -3623.559} C_VEL
LIN {X 0,Y 545.077,Z 115.395,A -85,B 0,C 180,E1 -3626.001,E2 -3626.001} C_VEL
LIN {X 0,Y 545.088,Z 115.401,A -85,B 0,C 180,E1 -3628.748,E2 -3628.748} C_VEL
LIN {X 0,Y 545.056,Z 115.398,A -85,B 0,C 180,E1 -3631.679,E2 -3631.679} C_VEL
LIN {X 0,Y 545.076,Z 115.403,A -85,B 0,C 180,E1 -3634.563,E2 -3634.563} C_VEL
LIN {X 0,Y 545.036,Z 115.401,A -85,B 0,C 180,E1 -3637.304,E2 -3637.304} C_VEL
LIN {X 0,Y 545.064,Z 115.402,A -85,B 0,C 180,E1 -3640.143,E2 -3640.143} C_VEL
LIN {X 0,Y 545.077,Z 115.396,A -85,B 0,C 180,E1 -3643.107,E2 -3643.107} C_VEL
LIN {X 0,Y 545.047,Z 115.408,A -85,B 0,C 180,E1 -3646.226,E2 -3646.226} C_VEL
LIN {X 0,Y 545.083,Z 115.395,A -85,B 0,C 180,E1 -3648.886,E2 -3648.886} C_VEL
LIN {X 0,Y 545.051,Z 115.404,A -85,B 0,C 180,E1 -3651.763,E2 -3651.763} C_VEL
LIN {X 0,Y 545.051,Z 115.4,A -85,B 0,C 180,E1 -3654.533,E2 -3654.533} C_VEL
LIN {X 0,Y 545.064,Z 115.399,A -85,B 0,C 180,E1 -3657.212,E2 -3657.212} C_VEL
LIN {X 0,Y 545.063,Z 115.404,A -85,B 0,C 180,E1 -3659.811,E2 -3659.811} C_VEL
LIN {X 0,Y 545.08,Z 115.395,A -85,B 0,C 180,E1 -3662.344,E2 -3662.344} C_VEL
LIN {X 0,Y 545.116,Z 115.392,A -85,B 0,C 180,E1 -3664.821,E2 -3664.821} C_VEL
LIN {X 0,Y 545.034,Z 115.392,A -85,B 0,C 180,E1 -3667.242,E2 -3667.242} C_VEL
LIN {X 0,Y 545.128,Z 115.589,A -85,B 0,C 180,E1 -3668.424,E2 -3668.424} C_VEL
LIN {X 0,Y 545.669,Z 119.838,A -85,B 0,C 180,E1 -3669.257,E2 -3669.257} C_VEL
LIN {X 0,Y 545.39,Z 136.278,A -85,B 0,C 180,E1 -3672.294,E2 -3672.294} C_VEL
LIN {X 0,Y 545.168,Z 151.452,A -85,B 0,C 180,E1 -3675.059,E2 -3675.059} C_VEL
LIN {X 0,Y 545.02,Z 168.289,A -85,B 0,C 180,E1 -3678.093,E2 -3678.093} C_VEL
LIN {X 0,Y 544.974,Z 171.106,A -85,B 0,C 180,E1 -3678.539,E2 -3678.539} C_VEL
LIN {X 0,Y 545.79,Z 179.003,A -85,B 0,C 180,E1 -3678.684,E2 -3678.684} C_VEL
LIN {X 0,Y 545.685,Z 246.874,A -85,B 0,C 180,E1 -3679.589,E2 -3679.589} C_VEL
LIN {X 0,Y 545.571,Z 256.145,A -85,B 0,C 180,E1 -3679.798,E2 -3679.798} C_VEL
LIN {X 0,Y 545.48,Z 264.623,A -85,B 0,C 180,E1 -3680.077,E2 -3680.077} C_VEL
LIN {X 0,Y 545.386,Z 273.136,A -85,B 0,C 180,E1 -3680.45,E2 -3680.45} C_VEL
LIN {X 0,Y 545.248,Z 281.479,A -85,B 0,C 180,E1 -3680.915,E2 -3680.915} C_VEL
LIN {X 0,Y 545.122,Z 289.529,A -85,B 0,C 180,E1 -3681.474,E2 -3681.474} C_VEL
LIN {X 0,Y 544.988,Z 298.218,A -85,B 0,C 180,E1 -3682.218,E2 -3682.218} C_VEL
LIN {X 0,Y 544.892,Z 306.743,A -85,B 0,C 180,E1 -3683.148,E2 -3683.148} C_VEL
LIN {X 0,Y 544.824,Z 313.431,A -85,B 0,C 180,E1 -3684.077,E2 -3684.077} C_VEL
LIN {X 0,Y 544.671,Z 317.82,A -85,B 0,C 180,E1 -3684.818,E2 -3684.818} C_VEL
LIN {X 0,Y 544.701,Z 322.997,A -85,B 0,C 180,E1 -3685.931,E2 -3685.931} C_VEL
LIN {X 0,Y 544.658,Z 326.796,A -85,B 0,C 180,E1 -3687.042,E2 -3687.042} C_VEL
LIN {X 0,Y 544.571,Z 328.542,A -85,B 0,C 180,E1 -3687.781,E2 -3687.781} C_VEL
LIN {X 0,Y 544.544,Z 329.794,A -85,B 0,C 180,E1 -3688.521,E2 -3688.521} C_VEL
LIN {X 0,Y 544.539,Z 330.574,A -85,B 0,C 180,E1 -3689.261,E2 -3689.261} C_VEL
LIN {X 0,Y 544.539,Z 330.869,A -85,B 0,C 180,E1 -3690,E2 -3690} C_VEL
LIN {X 0,Y 544.539,Z 330.573,A -85,B 0,C 180,E1 -3690.74,E2 -3690.74} C_VEL
LIN {X 0,Y 544.544,Z 329.793,A -85,B 0,C 180,E1 -3691.479,E2 -3691.479} C_VEL
LIN {X 0,Y 544.571,Z 328.54,A -85,B 0,C 180,E1 -3692.219,E2 -3692.219} C_VEL
LIN {X 0,Y 544.688,Z 325.64,A -85,B 0,C 180,E1 -3693.329,E2 -3693.329} C_VEL
LIN {X 0,Y 544.701,Z 322.995,A -85,B 0,C 180,E1 -3694.07,E2 -3694.07} C_VEL
LIN {X 0,Y 544.671,Z 317.815,A -85,B 0,C 180,E1 -3695.182,E2 -3695.182} C_VEL
LIN {X 0,Y 544.861,Z 311.779,A -85,B 0,C 180,E1 -3696.182,E2 -3696.182} C_VEL
LIN {X 0,Y 544.913,Z 305.233,A -85,B 0,C 180,E1 -3697.038,E2 -3697.038} C_VEL
LIN {X 0,Y 545.017,Z 297.198,A -85,B 0,C 180,E1 -3697.875,E2 -3697.875} C_VEL
LIN {X 0,Y 545.123,Z 289.529,A -85,B 0,C 180,E1 -3698.526,E2 -3698.526} C_VEL
LIN {X 0,Y 545.248,Z 281.474,A -85,B 0,C 180,E1 -3699.085,E2 -3699.085} C_VEL
LIN {X 0,Y 545.389,Z 273.131,A -85,B 0,C 180,E1 -3699.55,E2 -3699.55} C_VEL
LIN {X 0,Y 545.512,Z 264.617,A -85,B 0,C 180,E1 -3699.923,E2 -3699.923} C_VEL
LIN {X 0,Y 545.551,Z 255.302,A -85,B 0,C 180,E1 -3700.226,E2 -3700.226} C_VEL
LIN {X 0,Y 545.709,Z 244.26,A -85,B 0,C 180,E1 -3700.458,E2 -3700.458} C_VEL
LIN {X 0,Y 545.67,Z 176.819,A -85,B 0,C 180,E1 -3701.348,E2 -3701.348} C_VEL
LIN {X 0,Y 544.961,Z 171.036,A -85,B 0,C 180,E1 -3701.464,E2 -3701.464} C_VEL
LIN {X 0,Y 545.001,Z 165.129,A -85,B 0,C 180,E1 -3702.474,E2 -3702.474} C_VEL
LIN {X 0,Y 545.183,Z 149.34,A -85,B 0,C 180,E1 -3705.324,E2 -3705.324} C_VEL
LIN {X 0,Y 545.459,Z 133.541,A -85,B 0,C 180,E1 -3708.207,E2 -3708.207} C_VEL
LIN {X 0,Y 545.604,Z 118.78,A -85,B 0,C 180,E1 -3710.944,E2 -3710.944} C_VEL
LIN {X 0,Y 545.094,Z 115.457,A -85,B 0,C 180,E1 -3711.629,E2 -3711.629} C_VEL
LIN {X 0,Y 545.048,Z 115.393,A -85,B 0,C 180,E1 -3714.369,E2 -3714.369} C_VEL
LIN {X 0,Y 545.088,Z 115.395,A -85,B 0,C 180,E1 -3717.172,E2 -3717.172} C_VEL
LIN {X 0,Y 545.065,Z 115.397,A -85,B 0,C 180,E1 -3719.339,E2 -3719.339} C_VEL
LIN {X 0,Y 545.055,Z 115.402,A -85,B 0,C 180,E1 -3721.915,E2 -3721.915} C_VEL
LIN {X 0,Y 545.063,Z 115.4,A -85,B 0,C 180,E1 -3724.565,E2 -3724.565} C_VEL
LIN {X 0,Y 545.036,Z 115.401,A -85,B 0,C 180,E1 -3727.304,E2 -3727.304} C_VEL
LIN {X 0,Y 545.066,Z 115.403,A -85,B 0,C 180,E1 -3730.143,E2 -3730.143} C_VEL
LIN {X 0,Y 545.079,Z 115.396,A -85,B 0,C 180,E1 -3733.107,E2 -3733.107} C_VEL
LIN {X 0,Y 545.049,Z 115.401,A -85,B 0,C 180,E1 -3736.226,E2 -3736.226} C_VEL
LIN {X 0,Y 545.087,Z 115.395,A -85,B 0,C 180,E1 -3738.886,E2 -3738.886} C_VEL
LIN {X 0,Y 545.053,Z 115.404,A -85,B 0,C 180,E1 -3741.763,E2 -3741.763} C_VEL
LIN {X 0,Y 545.054,Z 115.398,A -85,B 0,C 180,E1 -3744.533,E2 -3744.533} C_VEL
LIN {X 0,Y 545.07,Z 115.404,A -85,B 0,C 180,E1 -3747.212,E2 -3747.212} C_VEL
LIN {X 0,Y 545.065,Z 115.398,A -85,B 0,C 180,E1 -3749.811,E2 -3749.811} C_VEL
LIN {X 0,Y 545.082,Z 115.395,A -85,B 0,C 180,E1 -3752.344,E2 -3752.344} C_VEL
LIN {X 0,Y 545.118,Z 115.396,A -85,B 0,C 180,E1 -3754.821,E2 -3754.821} C_VEL
LIN {X 0,Y 545.038,Z 115.405,A -85,B 0,C 180,E1 -3757.242,E2 -3757.242} C_VEL
LIN {X 0,Y 545.122,Z 115.393,A -85,B 0,C 180,E1 -3760.415,E2 -3760.415} C_VEL
LIN {X 0,Y 545.074,Z 115.396,A -85,B 0,C 180,E1 -3763.521,E2 -3763.521} C_VEL
LIN {X 0,Y 545.097,Z 115.393,A -85,B 0,C 180,E1 -3765.82,E2 -3765.82} C_VEL
LIN {X 0,Y 545.119,Z 115.394,A -85,B 0,C 180,E1 -3768.849,E2 -3768.849} C_VEL
LIN {X 0,Y 545.13,Z 115.391,A -85,B 0,C 180,E1 -3771.847,E2 -3771.847} C_VEL
LIN {X 0,Y 545.203,Z 115.381,A -85,B 0,C 180,E1 -3774.823,E2 -3774.823} C_VEL
LIN {X 0,Y 545.196,Z 115.384,A -85,B 0,C 180,E1 -3777.784,E2 -3777.784} C_VEL
LIN {X 0,Y 545.214,Z 115.379,A -85,B 0,C 180,E1 -3780.739,E2 -3780.739} C_VEL
LIN {X 0,Y 545.17,Z 115.384,A -85,B 0,C 180,E1 -3782.956,E2 -3782.956} C_VEL
LIN {X 0,Y 545.171,Z 115.392,A -85,B 0,C 180,E1 -3785.92,E2 -3785.92} C_VEL
LIN {X 0,Y 545.118,Z 115.39,A -85,B 0,C 180,E1 -3788.9,E2 -3788.9} C_VEL
LIN {X 0,Y 545.137,Z 115.393,A -85,B 0,C 180,E1 -3791.904,E2 -3791.904} C_VEL
LIN {X 0,Y 545.088,Z 115.396,A -85,B 0,C 180,E1 -3794.944,E2 -3794.944} C_VEL
LIN {X 0,Y 545.079,Z 115.396,A -85,B 0,C 180,E1 -3798.026,E2 -3798.026} C_VEL
LIN {X 0,Y 545.094,Z 115.393,A -85,B 0,C 180,E1 -3800.372,E2 -3800.372} C_VEL
LIN {X 0,Y 545.081,Z 115.399,A -85,B 0,C 180,E1 -3803.559,E2 -3803.559} C_VEL
LIN {X 0,Y 545.081,Z 115.395,A -85,B 0,C 180,E1 -3806.001,E2 -3806.001} C_VEL
LIN {X 0,Y 545.091,Z 115.399,A -85,B 0,C 180,E1 -3808.748,E2 -3808.748} C_VEL
LIN {X 0,Y 545.059,Z 115.398,A -85,B 0,C 180,E1 -3811.679,E2 -3811.679} C_VEL
LIN {X 0,Y 545.079,Z 115.401,A -85,B 0,C 180,E1 -3814.563,E2 -3814.563} C_VEL
LIN {X 0,Y 545.066,Z 115.401,A -85,B 0,C 180,E1 -3817.002,E2 -3817.002} C_VEL
LIN {X 0,Y 544.357,Z 115.488,A -85,B 0,C 180,E1 -3817.619,E2 -3817.619} C_VEL
LIN {X 0,Y 541.49,Z 115.851,A -85,B 0,C 180,E1 -3818.62,E2 -3818.62} C_VEL
LIN {X 0,Y 539.103,Z 116.143,A -85,B 0,C 180,E1 -3819.425,E2 -3819.425} C_VEL
LIN {X 0,Y 538.094,Z 116.267,A -85,B 0,C 180,E1 -3820.047,E2 -3820.047} C_VEL
LIN {X 0,Y 538.018,Z 116.275,A -85,B 0,C 180,E1 -3820.258,E2 -3820.258} C_VEL
LIN {X 0,Y 538.028,Z 116.275,A -85,B 0,C 180,E1 -3822.987,E2 -3822.987} C_VEL
LIN {X 0,Y 538.004,Z 116.283,A -85,B 0,C 180,E1 -3826.184,E2 -3826.184} C_VEL
LIN {X 0,Y 538.05,Z 116.271,A -85,B 0,C 180,E1 -3829.253,E2 -3829.253} C_VEL
LIN {X 0,Y 537.994,Z 116.287,A -85,B 0,C 180,E1 -3832.122,E2 -3832.122} C_VEL
LIN {X 0,Y 538.013,Z 116.275,A -85,B 0,C 180,E1 -3834.917,E2 -3834.917} C_VEL
LIN {X 0,Y 538.019,Z 116.279,A -85,B 0,C 180,E1 -3837.617,E2 -3837.617} C_VEL
LIN {X 0,Y 538.019,Z 116.277,A -85,B 0,C 180,E1 -3840.239,E2 -3840.239} C_VEL
LIN {X 0,Y 538.059,Z 116.269,A -85,B 0,C 180,E1 -3842.796,E2 -3842.796} C_VEL
LIN {X 0,Y 538.03,Z 116.277,A -85,B 0,C 180,E1 -3845.292,E2 -3845.292} C_VEL
LIN {X 0,Y 538.018,Z 116.279,A -85,B 0,C 180,E1 -3848.042,E2 -3848.042} C_VEL
LIN {X 0,Y 538.142,Z 116.445,A -85,B 0,C 180,E1 -3850.82,E2 -3850.82} C_VEL
LIN {X 0,Y 538.255,Z 124.29,A -85,B 0,C 180,E1 -3852.524,E2 -3852.524} C_VEL
LIN {X 0,Y 538.061,Z 138.947,A -85,B 0,C 180,E1 -3855.63,E2 -3855.63} C_VEL
LIN {X 0,Y 537.871,Z 152.291,A -85,B 0,C 180,E1 -3858.4,E2 -3858.4} C_VEL
LIN {X 0,Y 538.068,Z 154.049,A -85,B 0,C 180,E1 -3858.488,E2 -3858.488} C_VEL
LIN {X 0,Y 538.871,Z 161.158,A -85,B 0,C 180,E1 -3858.6,E2 -3858.6} C_VEL
LIN {X 0,Y 538.707,Z 227.701,A -85,B 0,C 180,E1 -3859.5,E2 -3859.5} C_VEL
LIN {X 0,Y 538.621,Z 236.922,A -85,B 0,C 180,E1 -3859.712,E2 -3859.712} C_VEL
LIN {X 0,Y 538.516,Z 246.574,A -85,B 0,C 180,E1 -3860.042,E2 -3860.042} C_VEL
LIN {X 0,Y 538.384,Z 256.65,A -85,B 0,C 180,E1 -3860.514,E2 -3860.514} C_VEL
LIN {X 0,Y 538.242,Z 267.109,A -85,B 0,C 180,E1 -3861.174,E2 -3861.174} C_VEL
LIN {X 0,Y 538.02,Z 275.269,A -85,B 0,C 180,E1 -3861.833,E2 -3861.833} C_VEL
LIN {X 0,Y 537.914,Z 282,A -85,B 0,C 180,E1 -3862.493,E2 -3862.493} C_VEL
LIN {X 0,Y 537.826,Z 288.608,A -85,B 0,C 180,E1 -3863.277,E2 -3863.277} C_VEL
LIN {X 0,Y 537.819,Z 293.664,A -85,B 0,C 180,E1 -3863.999,E2 -3863.999} C_VEL
LIN {X 0,Y 537.61,Z 298.088,A -85,B 0,C 180,E1 -3864.749,E2 -3864.749} C_VEL
LIN {X 0,Y 537.671,Z 301.769,A -85,B 0,C 180,E1 -3865.502,E2 -3865.502} C_VEL
LIN {X 0,Y 537.619,Z 305.956,A -85,B 0,C 180,E1 -3866.627,E2 -3866.627} C_VEL
LIN {X 0,Y 537.491,Z 308.883,A -85,B 0,C 180,E1 -3867.752,E2 -3867.752} C_VEL
LIN {X 0,Y 537.451,Z 310.166,A -85,B 0,C 180,E1 -3868.501,E2 -3868.501} C_VEL
LIN {X 0,Y 537.441,Z 310.981,A -85,B 0,C 180,E1 -3869.251,E2 -3869.251} C_VEL
LIN {X 0,Y 537.442,Z 311.29,A -85,B 0,C 180,E1 -3870,E2 -3870} C_VEL
LIN {X 0,Y 537.442,Z 311.019,A -85,B 0,C 180,E1 -3870.749,E2 -3870.749} C_VEL
LIN {X 0,Y 537.452,Z 310.283,A -85,B 0,C 180,E1 -3871.498,E2 -3871.498} C_VEL
LIN {X 0,Y 537.491,Z 309.078,A -85,B 0,C 180,E1 -3872.248,E2 -3872.248} C_VEL
LIN {X 0,Y 537.617,Z 306.233,A -85,B 0,C 180,E1 -3873.372,E2 -3873.372} C_VEL
LIN {X 0,Y 537.629,Z 303.647,A -85,B 0,C 180,E1 -3874.123,E2 -3874.123} C_VEL
LIN {X 0,Y 537.602,Z 298.549,A -85,B 0,C 180,E1 -3875.25,E2 -3875.25} C_VEL
LIN {X 0,Y 537.844,Z 292.799,A -85,B 0,C 180,E1 -3876.23,E2 -3876.23} C_VEL
LIN {X 0,Y 537.862,Z 286.179,A -85,B 0,C 180,E1 -3877.13,E2 -3877.13} C_VEL
LIN {X 0,Y 537.992,Z 277.257,A -85,B 0,C 180,E1 -3878.073,E2 -3878.073} C_VEL
LIN {X 0,Y 538.176,Z 269.508,A -85,B 0,C 180,E1 -3878.732,E2 -3878.732} C_VEL
LIN {X 0,Y 538.281,Z 261.34,A -85,B 0,C 180,E1 -3879.298,E2 -3879.298} C_VEL
LIN {X 0,Y 538.435,Z 252.82,A -85,B 0,C 180,E1 -3879.769,E2 -3879.769} C_VEL
LIN {X 0,Y 538.595,Z 242.829,A -85,B 0,C 180,E1 -3880.193,E2 -3880.193} C_VEL
LIN {X 0,Y 538.751,Z 231.334,A -85,B 0,C 180,E1 -3880.523,E2 -3880.523} C_VEL
LIN {X 0,Y 538.782,Z 212.587,A -85,B 0,C 180,E1 -3880.807,E2 -3880.807} C_VEL
LIN {X 0,Y 538.769,Z 158.741,A -85,B 0,C 180,E1 -3881.524,E2 -3881.524} C_VEL
LIN {X 0,Y 537.919,Z 152.895,A -85,B 0,C 180,E1 -3881.64,E2 -3881.64} C_VEL
LIN {X 0,Y 537.897,Z 151.861,A -85,B 0,C 180,E1 -3881.763,E2 -3881.763} C_VEL
LIN {X 0,Y 538.072,Z 137.039,A -85,B 0,C 180,E1 -3884.862,E2 -3884.862} C_VEL
LIN {X 0,Y 538.29,Z 123.011,A -85,B 0,C 180,E1 -3887.84,E2 -3887.84} C_VEL
LIN {X 0,Y 538.131,Z 116.372,A -85,B 0,C 180,E1 -3889.304,E2 -3889.304} C_VEL
LIN {X 0,Y 537.993,Z 116.285,A -85,B 0,C 180,E1 -3892.261,E2 -3892.261} C_VEL
LIN {X 0,Y 538.071,Z 116.268,A -85,B 0,C 180,E1 -3895.533,E2 -3895.533} C_VEL
LIN {X 0,Y 538.041,Z 116.276,A -85,B 0,C 180,E1 -3898.05,E2 -3898.05} C_VEL
LIN {X 0,Y 538.021,Z 116.278,A -85,B 0,C 180,E1 -3900.627,E2 -3900.627} C_VEL
LIN {X 0,Y 538.019,Z 116.275,A -85,B 0,C 180,E1 -3903.278,E2 -3903.278} C_VEL
LIN {X 0,Y 538.023,Z 116.283,A -85,B 0,C 180,E1 -3906.002,E2 -3906.002} C_VEL
LIN {X 0,Y 538.013,Z 116.275,A -85,B 0,C 180,E1 -3908.83,E2 -3908.83} C_VEL
LIN {X 0,Y 538.03,Z 116.282,A -85,B 0,C 180,E1 -3911.773,E2 -3911.773} C_VEL
LIN {X 0,Y 538.006,Z 116.276,A -85,B 0,C 180,E1 -3914.862,E2 -3914.862} C_VEL
LIN {X 0,Y 538.033,Z 116.275,A -85,B 0,C 180,E1 -3918.121,E2 -3918.121} C_VEL
LIN {X 0,Y 538.033,Z 116.273,A -85,B 0,C 180,E1 -3920.415,E2 -3920.415} C_VEL
LIN {X 0,Y 538.027,Z 116.278,A -85,B 0,C 180,E1 -3923.067,E2 -3923.067} C_VEL
LIN {X 0,Y 538.023,Z 116.276,A -85,B 0,C 180,E1 -3925.827,E2 -3925.827} C_VEL
LIN {X 0,Y 538.008,Z 116.277,A -85,B 0,C 180,E1 -3928.498,E2 -3928.498} C_VEL
LIN {X 0,Y 538.059,Z 116.279,A -85,B 0,C 180,E1 -3931.1,E2 -3931.1} C_VEL
LIN {X 0,Y 538.04,Z 116.273,A -85,B 0,C 180,E1 -3933.633,E2 -3933.633} C_VEL
LIN {X 0,Y 538.006,Z 116.277,A -85,B 0,C 180,E1 -3936.122,E2 -3936.122} C_VEL
LIN {X 0,Y 538.039,Z 116.274,A -85,B 0,C 180,E1 -3939.349,E2 -3939.349} C_VEL
LIN {X 0,Y 538.053,Z 116.277,A -85,B 0,C 180,E1 -3942.517,E2 -3942.517} C_VEL
LIN {X 0,Y 538.063,Z 116.269,A -85,B 0,C 180,E1 -3945.631,E2 -3945.631} C_VEL
LIN {X 0,Y 538.076,Z 116.272,A -85,B 0,C 180,E1 -3948.701,E2 -3948.701} C_VEL
LIN {X 0,Y 538.085,Z 116.268,A -85,B 0,C 180,E1 -3951.739,E2 -3951.739} C_VEL
LIN {X 0,Y 538.161,Z 116.259,A -85,B 0,C 180,E1 -3954.755,E2 -3954.755} C_VEL
LIN {X 0,Y 538.169,Z 116.26,A -85,B 0,C 180,E1 -3957.755,E2 -3957.755} C_VEL
LIN {X 0,Y 538.182,Z 116.255,A -85,B 0,C 180,E1 -3960.748,E2 -3960.748} C_VEL
LIN {X 0,Y 538.136,Z 116.26,A -85,B 0,C 180,E1 -3962.994,E2 -3962.994} C_VEL
LIN {X 0,Y 538.123,Z 116.267,A -85,B 0,C 180,E1 -3965.997,E2 -3965.997} C_VEL
LIN {X 0,Y 538.067,Z 116.27,A -85,B 0,C 180,E1 -3969.018,E2 -3969.018} C_VEL
LIN {X 0,Y 538.082,Z 116.269,A -85,B 0,C 180,E1 -3972.062,E2 -3972.062} C_VEL
LIN {X 0,Y 538.044,Z 116.277,A -85,B 0,C 180,E1 -3975.144,E2 -3975.144} C_VEL
LIN {X 0,Y 538.03,Z 116.273,A -85,B 0,C 180,E1 -3978.27,E2 -3978.27} C_VEL
LIN {X 0,Y 538.038,Z 116.274,A -85,B 0,C 180,E1 -3980.651,E2 -3980.651} C_VEL
LIN {X 0,Y 538.001,Z 116.277,A -85,B 0,C 180,E1 -3983.888,E2 -3983.888} C_VEL
LIN {X 0,Y 538.04,Z 116.273,A -85,B 0,C 180,E1 -3986.367,E2 -3986.367} C_VEL
LIN {X 0,Y 538.029,Z 116.281,A -85,B 0,C 180,E1 -3988.934,E2 -3988.934} C_VEL
LIN {X 0,Y 538.008,Z 116.276,A -85,B 0,C 180,E1 -3991.887,E2 -3991.887} C_VEL
LIN {X 0,Y 538.025,Z 116.283,A -85,B 0,C 180,E1 -3994.62,E2 -3994.62} C_VEL
LIN {X 0,Y 538.005,Z 116.278,A -85,B 0,C 180,E1 -3997.17,E2 -3997.17} C_VEL
LIN {X 0,Y 538.021,Z 116.275,A -85,B 0,C 180,E1 -3999.797,E2 -3999.797} C_VEL
LIN {X 0,Y 538.017,Z 116.278,A -85,B 0,C 180,E1 -4002.786,E2 -4002.786} C_VEL
LIN {X 0,Y 538.005,Z 116.276,A -85,B 0,C 180,E1 -4005.138,E2 -4005.138} C_VEL
LIN {X 0,Y 538.033,Z 116.28,A -85,B 0,C 180,E1 -4008.227,E2 -4008.227} C_VEL
LIN {X 0,Y 538.011,Z 116.276,A -85,B 0,C 180,E1 -4011.17,E2 -4011.17} C_VEL
LIN {X 0,Y 538.022,Z 116.28,A -85,B 0,C 180,E1 -4014.085,E2 -4014.085} C_VEL
LIN {X 0,Y 538.029,Z 116.273,A -85,B 0,C 180,E1 -4016.728,E2 -4016.728} C_VEL
LIN {X 0,Y 538.025,Z 116.281,A -85,B 0,C 180,E1 -4019.556,E2 -4019.556} C_VEL
LIN {X 0,Y 538.039,Z 116.276,A -85,B 0,C 180,E1 -4021.95,E2 -4021.95} C_VEL
LIN {X 0,Y 538.07,Z 116.269,A -85,B 0,C 180,E1 -4024.467,E2 -4024.467} C_VEL
LIN {X 0,Y 537.992,Z 116.274,A -85,B 0,C 180,E1 -4027.739,E2 -4027.739} C_VEL
LIN {X 0,Y 538.079,Z 116.526,A -85,B 0,C 180,E1 -4028.332,E2 -4028.332} C_VEL
LIN {X 0,Y 538.69,Z 120.783,A -85,B 0,C 180,E1 -4029.175,E2 -4029.175} C_VEL
LIN {X 0,Y 538.387,Z 136.451,A -85,B 0,C 180,E1 -4032.11,E2 -4032.11} C_VEL
LIN {X 0,Y 538.126,Z 152.729,A -85,B 0,C 180,E1 -4035.116,E2 -4035.116} C_VEL
LIN {X 0,Y 537.931,Z 169.873,A -85,B 0,C 180,E1 -4038.244,E2 -4038.244} C_VEL
LIN {X 0,Y 537.928,Z 171.018,A -85,B 0,C 180,E1 -4038.39,E2 -4038.39} C_VEL
LIN {X 0,Y 538.849,Z 179.136,A -85,B 0,C 180,E1 -4038.539,E2 -4038.539} C_VEL
LIN {X 0,Y 538.716,Z 246.746,A -85,B 0,C 180,E1 -4039.453,E2 -4039.453} C_VEL
LIN {X 0,Y 538.598,Z 256.017,A -85,B 0,C 180,E1 -4039.664,E2 -4039.664} C_VEL
LIN {X 0,Y 538.484,Z 264.494,A -85,B 0,C 180,E1 -4039.947,E2 -4039.947} C_VEL
LIN {X 0,Y 538.387,Z 273.007,A -85,B 0,C 180,E1 -4040.325,E2 -4040.325} C_VEL
LIN {X 0,Y 538.24,Z 281.351,A -85,B 0,C 180,E1 -4040.796,E2 -4040.796} C_VEL
LIN {X 0,Y 538.089,Z 289.401,A -85,B 0,C 180,E1 -4041.362,E2 -4041.362} C_VEL
LIN {X 0,Y 537.951,Z 298.089,A -85,B 0,C 180,E1 -4042.116,E2 -4042.116} C_VEL
LIN {X 0,Y 537.824,Z 306.614,A -85,B 0,C 180,E1 -4043.058,E2 -4043.058} C_VEL
LIN {X 0,Y 537.757,Z 313.302,A -85,B 0,C 180,E1 -4043.999,E2 -4043.999} C_VEL
LIN {X 0,Y 537.603,Z 317.691,A -85,B 0,C 180,E1 -4044.75,E2 -4044.75} C_VEL
LIN {X 0,Y 537.623,Z 322.868,A -85,B 0,C 180,E1 -4045.877,E2 -4045.877} C_VEL
LIN {X 0,Y 537.562,Z 326.667,A -85,B 0,C 180,E1 -4047.003,E2 -4047.003} C_VEL
LIN {X 0,Y 537.49,Z 328.414,A -85,B 0,C 180,E1 -4047.752,E2 -4047.752} C_VEL
LIN {X 0,Y 537.45,Z 329.665,A -85,B 0,C 180,E1 -4048.502,E2 -4048.502} C_VEL
LIN {X 0,Y 537.44,Z 330.445,A -85,B 0,C 180,E1 -4049.251,E2 -4049.251} C_VEL
LIN {X 0,Y 537.441,Z 330.74,A -85,B 0,C 180,E1 -4050,E2 -4050} C_VEL
LIN {X 0,Y 537.44,Z 330.445,A -85,B 0,C 180,E1 -4050.749,E2 -4050.749} C_VEL
LIN {X 0,Y 537.45,Z 329.664,A -85,B 0,C 180,E1 -4051.499,E2 -4051.499} C_VEL
LIN {X 0,Y 537.49,Z 328.412,A -85,B 0,C 180,E1 -4052.248,E2 -4052.248} C_VEL
LIN {X 0,Y 537.588,Z 325.511,A -85,B 0,C 180,E1 -4053.373,E2 -4053.373} C_VEL
LIN {X 0,Y 537.623,Z 322.866,A -85,B 0,C 180,E1 -4054.123,E2 -4054.123} C_VEL
LIN {X 0,Y 537.604,Z 317.687,A -85,B 0,C 180,E1 -4055.251,E2 -4055.251} C_VEL
LIN {X 0,Y 537.783,Z 311.959,A -85,B 0,C 180,E1 -4056.215,E2 -4056.215} C_VEL
LIN {X 0,Y 537.848,Z 305.105,A -85,B 0,C 180,E1 -4057.131,E2 -4057.131} C_VEL
LIN {X 0,Y 537.943,Z 297.069,A -85,B 0,C 180,E1 -4057.979,E2 -4057.979} C_VEL
LIN {X 0,Y 538.089,Z 289.4,A -85,B 0,C 180,E1 -4058.639,E2 -4058.639} C_VEL
LIN {X 0,Y 538.241,Z 281.346,A -85,B 0,C 180,E1 -4059.204,E2 -4059.204} C_VEL
LIN {X 0,Y 538.378,Z 273.002,A -85,B 0,C 180,E1 -4059.676,E2 -4059.676} C_VEL
LIN {X 0,Y 538.524,Z 264.489,A -85,B 0,C 180,E1 -4060.053,E2 -4060.053} C_VEL
LIN {X 0,Y 538.569,Z 255.174,A -85,B 0,C 180,E1 -4060.36,E2 -4060.36} C_VEL
LIN {X 0,Y 538.726,Z 244.131,A -85,B 0,C 180,E1 -4060.595,E2 -4060.595} C_VEL
LIN {X 0,Y 538.715,Z 177.227,A -85,B 0,C 180,E1 -4061.489,E2 -4061.489} C_VEL
LIN {X 0,Y 537.943,Z 171.195,A -85,B 0,C 180,E1 -4061.599,E2 -4061.599} C_VEL
LIN {X 0,Y 537.932,Z 169.873,A -85,B 0,C 180,E1 -4061.756,E2 -4061.756} C_VEL
LIN {X 0,Y 538.127,Z 152.726,A -85,B 0,C 180,E1 -4064.884,E2 -4064.884} C_VEL
LIN {X 0,Y 538.388,Z 136.446,A -85,B 0,C 180,E1 -4067.891,E2 -4067.891} C_VEL
LIN {X 0,Y 538.685,Z 120.782,A -85,B 0,C 180,E1 -4070.825,E2 -4070.825} C_VEL
LIN {X 0,Y 538.033,Z 116.326,A -85,B 0,C 180,E1 -4071.742,E2 -4071.742} C_VEL
LIN {X 0,Y 538.043,Z 116.272,A -85,B 0,C 180,E1 -4074.708,E2 -4074.708} C_VEL
LIN {X 0,Y 538.053,Z 116.27,A -85,B 0,C 180,E1 -4077.351,E2 -4077.351} C_VEL
LIN {X 0,Y 538.017,Z 116.276,A -85,B 0,C 180,E1 -4079.761,E2 -4079.761} C_VEL
LIN {X 0,Y 538.018,Z 116.282,A -85,B 0,C 180,E1 -4082.383,E2 -4082.383} C_VEL
LIN {X 0,Y 537.999,Z 116.277,A -85,B 0,C 180,E1 -4085.084,E2 -4085.084} C_VEL
LIN {X 0,Y 537.993,Z 116.285,A -85,B 0,C 180,E1 -4087.878,E2 -4087.878} C_VEL
LIN {X 0,Y 538.048,Z 116.271,A -85,B 0,C 180,E1 -4090.776,E2 -4090.776} C_VEL
LIN {X 0,Y 538.003,Z 116.286,A -85,B 0,C 180,E1 -4093.816,E2 -4093.816} C_VEL
LIN {X 0,Y 538.027,Z 116.274,A -85,B 0,C 180,E1 -4097.013,E2 -4097.013} C_VEL
LIN {X 0,Y 538.049,Z 116.275,A -85,B 0,C 180,E1 -4099.253,E2 -4099.253} C_VEL
LIN {X 0,Y 537.993,Z 116.279,A -85,B 0,C 180,E1 -4102.122,E2 -4102.122} C_VEL
LIN {X 0,Y 538.013,Z 116.278,A -85,B 0,C 180,E1 -4104.917,E2 -4104.917} C_VEL
LIN {X 0,Y 538.02,Z 116.279,A -85,B 0,C 180,E1 -4107.617,E2 -4107.617} C_VEL
LIN {X 0,Y 538.018,Z 116.275,A -85,B 0,C 180,E1 -4110.239,E2 -4110.239} C_VEL
LIN {X 0,Y 538.058,Z 116.274,A -85,B 0,C 180,E1 -4112.796,E2 -4112.796} C_VEL
LIN {X 0,Y 538.048,Z 116.276,A -85,B 0,C 180,E1 -4115.293,E2 -4115.293} C_VEL
LIN {X 0,Y 538.024,Z 116.278,A -85,B 0,C 180,E1 -4118.546,E2 -4118.546} C_VEL
LIN {X 0,Y 538.039,Z 116.279,A -85,B 0,C 180,E1 -4120.94,E2 -4120.94} C_VEL
LIN {X 0,Y 538.026,Z 116.275,A -85,B 0,C 180,E1 -4123.299,E2 -4123.299} C_VEL
LIN {X 0,Y 538.066,Z 116.269,A -85,B 0,C 180,E1 -4125.631,E2 -4125.631} C_VEL
LIN {X 0,Y 538.079,Z 116.273,A -85,B 0,C 180,E1 -4128.702,E2 -4128.702} C_VEL
LIN {X 0,Y 538.087,Z 116.267,A -85,B 0,C 180,E1 -4131.74,E2 -4131.74} C_VEL
LIN {X 0,Y 538.161,Z 116.259,A -85,B 0,C 180,E1 -4134.755,E2 -4134.755} C_VEL
LIN {X 0,Y 538.168,Z 116.259,A -85,B 0,C 180,E1 -4137.755,E2 -4137.755} C_VEL
LIN {X 0,Y 538.184,Z 116.255,A -85,B 0,C 180,E1 -4140.748,E2 -4140.748} C_VEL
LIN {X 0,Y 538.137,Z 116.26,A -85,B 0,C 180,E1 -4142.995,E2 -4142.995} C_VEL
LIN {X 0,Y 538.125,Z 116.268,A -85,B 0,C 180,E1 -4145.997,E2 -4145.997} C_VEL
LIN {X 0,Y 538.07,Z 116.269,A -85,B 0,C 180,E1 -4149.018,E2 -4149.018} C_VEL
LIN {X 0,Y 538.085,Z 116.269,A -85,B 0,C 180,E1 -4152.063,E2 -4152.063} C_VEL
LIN {X 0,Y 538.047,Z 116.275,A -85,B 0,C 180,E1 -4155.144,E2 -4155.144} C_VEL
LIN {X 0,Y 538.031,Z 116.273,A -85,B 0,C 180,E1 -4158.27,E2 -4158.27} C_VEL
LIN {X 0,Y 538.039,Z 116.273,A -85,B 0,C 180,E1 -4160.651,E2 -4160.651} C_VEL
LIN {X 0,Y 538.004,Z 116.277,A -85,B 0,C 180,E1 -4163.888,E2 -4163.888} C_VEL
LIN {X 0,Y 538.043,Z 116.272,A -85,B 0,C 180,E1 -4166.367,E2 -4166.367} C_VEL
LIN {X 0,Y 538.033,Z 116.281,A -85,B 0,C 180,E1 -4168.934,E2 -4168.934} C_VEL
LIN {X 0,Y 538.012,Z 116.275,A -85,B 0,C 180,E1 -4171.887,E2 -4171.887} C_VEL
LIN {X 0,Y 538.029,Z 116.28,A -85,B 0,C 180,E1 -4174.62,E2 -4174.62} C_VEL
LIN {X 0,Y 538.008,Z 116.278,A -85,B 0,C 180,E1 -4177.17,E2 -4177.17} C_VEL
LIN {X 0,Y 538.018,Z 116.275,A -85,B 0,C 180,E1 -4180.258,E2 -4180.258} C_VEL
LIN {X 0,Y 537.369,Z 116.361,A -85,B 0,C 180,E1 -4180.883,E2 -4180.883} C_VEL
LIN {X 0,Y 534.517,Z 116.713,A -85,B 0,C 180,E1 -4181.898,E2 -4181.898} C_VEL
LIN {X 0,Y 532.091,Z 117.018,A -85,B 0,C 180,E1 -4182.715,E2 -4182.715} C_VEL
LIN {X 0,Y 531.041,Z 117.144,A -85,B 0,C 180,E1 -4183.346,E2 -4183.346} C_VEL
LIN {X 0,Y 530.953,Z 117.155,A -85,B 0,C 180,E1 -4183.56,E2 -4183.56} C_VEL
LIN {X 0,Y 530.956,Z 117.161,A -85,B 0,C 180,E1 -4186.504,E2 -4186.504} C_VEL
LIN {X 0,Y 530.985,Z 117.151,A -85,B 0,C 180,E1 -4188.977,E2 -4188.977} C_VEL
LIN {X 0,Y 530.958,Z 117.156,A -85,B 0,C 180,E1 -4191.529,E2 -4191.529} C_VEL
LIN {X 0,Y 530.978,Z 117.155,A -85,B 0,C 180,E1 -4194.382,E2 -4194.382} C_VEL
LIN {X 0,Y 530.968,Z 117.153,A -85,B 0,C 180,E1 -4197.133,E2 -4197.133} C_VEL
LIN {X 0,Y 530.972,Z 117.161,A -85,B 0,C 180,E1 -4199.803,E2 -4199.803} C_VEL
LIN {X 0,Y 531.015,Z 117.148,A -85,B 0,C 180,E1 -4202.467,E2 -4202.467} C_VEL
LIN {X 0,Y 530.997,Z 117.15,A -85,B 0,C 180,E1 -4204.942,E2 -4204.942} C_VEL
LIN {X 0,Y 530.974,Z 117.156,A -85,B 0,C 180,E1 -4208.247,E2 -4208.247} C_VEL
LIN {X 0,Y 531.071,Z 117.279,A -85,B 0,C 180,E1 -4210.73,E2 -4210.73} C_VEL
LIN {X 0,Y 531.246,Z 124.304,A -85,B 0,C 180,E1 -4212.285,E2 -4212.285} C_VEL
LIN {X 0,Y 531.008,Z 138.977,A -85,B 0,C 180,E1 -4215.435,E2 -4215.435} C_VEL
LIN {X 0,Y 530.848,Z 152.483,A -85,B 0,C 180,E1 -4218.254,E2 -4218.254} C_VEL
LIN {X 0,Y 531.045,Z 154.192,A -85,B 0,C 180,E1 -4218.333,E2 -4218.333} C_VEL
LIN {X 0,Y 531.924,Z 160.74,A -85,B 0,C 180,E1 -4218.441,E2 -4218.441} C_VEL
LIN {X 0,Y 531.736,Z 227.862,A -85,B 0,C 180,E1 -4219.361,E2 -4219.361} C_VEL
LIN {X 0,Y 531.657,Z 237.07,A -85,B 0,C 180,E1 -4219.576,E2 -4219.576} C_VEL
LIN {X 0,Y 531.549,Z 246.716,A -85,B 0,C 180,E1 -4219.91,E2 -4219.91} C_VEL
LIN {X 0,Y 531.403,Z 256.79,A -85,B 0,C 180,E1 -4220.388,E2 -4220.388} C_VEL
LIN {X 0,Y 531.233,Z 267.245,A -85,B 0,C 180,E1 -4221.057,E2 -4221.057} C_VEL
LIN {X 0,Y 530.996,Z 275.404,A -85,B 0,C 180,E1 -4221.724,E2 -4221.724} C_VEL
LIN {X 0,Y 530.864,Z 282.133,A -85,B 0,C 180,E1 -4222.392,E2 -4222.392} C_VEL
LIN {X 0,Y 530.774,Z 289.239,A -85,B 0,C 180,E1 -4223.255,E2 -4223.255} C_VEL
LIN {X 0,Y 530.723,Z 294.965,A -85,B 0,C 180,E1 -4224.109,E2 -4224.109} C_VEL
LIN {X 0,Y 530.528,Z 300.126,A -85,B 0,C 180,E1 -4225.06,E2 -4225.06} C_VEL
LIN {X 0,Y 530.527,Z 304.904,A -85,B 0,C 180,E1 -4226.202,E2 -4226.202} C_VEL
LIN {X 0,Y 530.498,Z 307.233,A -85,B 0,C 180,E1 -4226.962,E2 -4226.962} C_VEL
LIN {X 0,Y 530.413,Z 309.011,A -85,B 0,C 180,E1 -4227.722,E2 -4227.722} C_VEL
LIN {X 0,Y 530.36,Z 310.295,A -85,B 0,C 180,E1 -4228.481,E2 -4228.481} C_VEL
LIN {X 0,Y 530.343,Z 311.109,A -85,B 0,C 180,E1 -4229.241,E2 -4229.241} C_VEL
LIN {X 0,Y 530.344,Z 311.418,A -85,B 0,C 180,E1 -4230,E2 -4230} C_VEL
LIN {X 0,Y 530.344,Z 311.147,A -85,B 0,C 180,E1 -4230.759,E2 -4230.759} C_VEL
LIN {X 0,Y 530.361,Z 310.41,A -85,B 0,C 180,E1 -4231.518,E2 -4231.518} C_VEL
LIN {X 0,Y 530.413,Z 309.204,A -85,B 0,C 180,E1 -4232.278,E2 -4232.278} C_VEL
LIN {X 0,Y 530.519,Z 306.359,A -85,B 0,C 180,E1 -4233.417,E2 -4233.417} C_VEL
LIN {X 0,Y 530.56,Z 303.772,A -85,B 0,C 180,E1 -4234.178,E2 -4234.178} C_VEL
LIN {X 0,Y 530.541,Z 298.674,A -85,B 0,C 180,E1 -4235.32,E2 -4235.32} C_VEL
LIN {X 0,Y 530.789,Z 293.127,A -85,B 0,C 180,E1 -4236.28,E2 -4236.28} C_VEL
LIN {X 0,Y 530.811,Z 286.302,A -85,B 0,C 180,E1 -4237.226,E2 -4237.226} C_VEL
LIN {X 0,Y 530.979,Z 277.377,A -85,B 0,C 180,E1 -4238.18,E2 -4238.18} C_VEL
LIN {X 0,Y 531.167,Z 269.627,A -85,B 0,C 180,E1 -4238.848,E2 -4238.848} C_VEL
LIN {X 0,Y 531.281,Z 261.458,A -85,B 0,C 180,E1 -4239.422,E2 -4239.422} C_VEL
LIN {X 0,Y 531.449,Z 252.936,A -85,B 0,C 180,E1 -4239.899,E2 -4239.899} C_VEL
LIN {X 0,Y 531.633,Z 241.691,A -85,B 0,C 180,E1 -4240.376,E2 -4240.376} C_VEL
LIN {X 0,Y 531.803,Z 230.131,A -85,B 0,C 180,E1 -4240.686,E2 -4240.686} C_VEL
LIN {X 0,Y 531.843,Z 205.517,A -85,B 0,C 180,E1 -4241.046,E2 -4241.046} C_VEL
LIN {X 0,Y 531.757,Z 158.939,A -85,B 0,C 180,E1 -4241.677,E2 -4241.677} C_VEL
LIN {X 0,Y 530.885,Z 152.853,A -85,B 0,C 180,E1 -4241.804,E2 -4241.804} C_VEL
LIN {X 0,Y 530.845,Z 152.072,A -85,B 0,C 180,E1 -4241.896,E2 -4241.896} C_VEL
LIN {X 0,Y 531.033,Z 137.562,A -85,B 0,C 180,E1 -4244.956,E2 -4244.956} C_VEL
LIN {X 0,Y 531.267,Z 123.071,A -85,B 0,C 180,E1 -4248.072,E2 -4248.072} C_VEL
LIN {X 0,Y 531.099,Z 117.243,A -85,B 0,C 180,E1 -4249.387,E2 -4249.387} C_VEL
LIN {X 0,Y 530.945,Z 117.165,A -85,B 0,C 180,E1 -4252.573,E2 -4252.573} C_VEL
LIN {X 0,Y 530.995,Z 117.151,A -85,B 0,C 180,E1 -4255.058,E2 -4255.058} C_VEL
LIN {X 0,Y 531.014,Z 117.148,A -85,B 0,C 180,E1 -4257.595,E2 -4257.595} C_VEL
LIN {X 0,Y 530.974,Z 117.155,A -85,B 0,C 180,E1 -4260.645,E2 -4260.645} C_VEL
LIN {X 0,Y 530.96,Z 117.158,A -85,B 0,C 180,E1 -4263.774,E2 -4263.774} C_VEL
LIN {X 0,Y 530.966,Z 117.155,A -85,B 0,C 180,E1 -4266.557,E2 -4266.557} C_VEL
LIN {X 0,Y 530.978,Z 117.16,A -85,B 0,C 180,E1 -4269.853,E2 -4269.853} C_VEL
LIN {X 0,Y 530.977,Z 117.153,A -85,B 0,C 180,E1 -4272.456,E2 -4272.456} C_VEL
LIN {X 0,Y 530.977,Z 117.16,A -85,B 0,C 180,E1 -4275.622,E2 -4275.622} C_VEL
LIN {X 0,Y 530.996,Z 117.149,A -85,B 0,C 180,E1 -4278.564,E2 -4278.564} C_VEL
LIN {X 0,Y 530.957,Z 117.162,A -85,B 0,C 180,E1 -4281.529,E2 -4281.529} C_VEL
LIN {X 0,Y 530.976,Z 117.152,A -85,B 0,C 180,E1 -4284.382,E2 -4284.382} C_VEL
LIN {X 0,Y 530.966,Z 117.161,A -85,B 0,C 180,E1 -4287.133,E2 -4287.133} C_VEL
LIN {X 0,Y 530.968,Z 117.154,A -85,B 0,C 180,E1 -4289.803,E2 -4289.803} C_VEL
LIN {X 0,Y 531.011,Z 117.149,A -85,B 0,C 180,E1 -4292.467,E2 -4292.467} C_VEL
LIN {X 0,Y 531.004,Z 117.158,A -85,B 0,C 180,E1 -4294.942,E2 -4294.942} C_VEL
LIN {X 0,Y 530.97,Z 117.154,A -85,B 0,C 180,E1 -4298.247,E2 -4298.247} C_VEL
LIN {X 0,Y 530.995,Z 117.158,A -85,B 0,C 180,E1 -4300.677,E2 -4300.677} C_VEL
LIN {X 0,Y 530.985,Z 117.154,A -85,B 0,C 180,E1 -4303.071,E2 -4303.071} C_VEL
LIN {X 0,Y 531.018,Z 117.147,A -85,B 0,C 180,E1 -4305.436,E2 -4305.436} C_VEL
LIN {X 0,Y 531.048,Z 117.15,A -85,B 0,C 180,E1 -4308.55,E2 -4308.55} C_VEL
LIN {X 0,Y 531.054,Z 117.143,A -85,B 0,C 180,E1 -4311.629,E2 -4311.629} C_VEL
LIN {X 0,Y 531.12,Z 117.136,A -85,B 0,C 180,E1 -4314.685,E2 -4314.685} C_VEL
LIN {X 0,Y 531.14,Z 117.136,A -85,B 0,C 180,E1 -4317.725,E2 -4317.725} C_VEL
LIN {X 0,Y 531.152,Z 117.13,A -85,B 0,C 180,E1 -4320.758,E2 -4320.758} C_VEL
LIN {X 0,Y 531.103,Z 117.136,A -85,B 0,C 180,E1 -4323.034,E2 -4323.034} C_VEL
LIN {X 0,Y 531.083,Z 117.143,A -85,B 0,C 180,E1 -4326.077,E2 -4326.077} C_VEL
LIN {X 0,Y 531.027,Z 117.148,A -85,B 0,C 180,E1 -4329.138,E2 -4329.138} C_VEL
LIN {X 0,Y 531.04,Z 117.145,A -85,B 0,C 180,E1 -4332.225,E2 -4332.225} C_VEL
LIN {X 0,Y 530.994,Z 117.158,A -85,B 0,C 180,E1 -4335.35,E2 -4335.35} C_VEL
LIN {X 0,Y 530.99,Z 117.151,A -85,B 0,C 180,E1 -4338.521,E2 -4338.521} C_VEL
LIN {X 0,Y 530.999,Z 117.154,A -85,B 0,C 180,E1 -4340.938,E2 -4340.938} C_VEL
LIN {X 0,Y 530.969,Z 117.153,A -85,B 0,C 180,E1 -4344.225,E2 -4344.225} C_VEL
LIN {X 0,Y 531,Z 117.155,A -85,B 0,C 180,E1 -4346.744,E2 -4346.744} C_VEL
LIN {X 0,Y 530.98,Z 117.154,A -85,B 0,C 180,E1 -4349.323,E2 -4349.323} C_VEL
LIN {X 0,Y 530.964,Z 117.155,A -85,B 0,C 180,E1 -4352.1,E2 -4352.1} C_VEL
LIN {X 0,Y 530.982,Z 117.157,A -85,B 0,C 180,E1 -4354.853,E2 -4354.853} C_VEL
LIN {X 0,Y 530.964,Z 117.153,A -85,B 0,C 180,E1 -4357.508,E2 -4357.508} C_VEL
LIN {X 0,Y 530.979,Z 117.161,A -85,B 0,C 180,E1 -4360.433,E2 -4360.433} C_VEL
LIN {X 0,Y 530.963,Z 117.154,A -85,B 0,C 180,E1 -4363.495,E2 -4363.495} C_VEL
LIN {X 0,Y 530.953,Z 117.159,A -85,B 0,C 180,E1 -4366.505,E2 -4366.505} C_VEL
LIN {X 0,Y 530.984,Z 117.151,A -85,B 0,C 180,E1 -4368.976,E2 -4368.976} C_VEL
LIN {X 0,Y 530.955,Z 117.157,A -85,B 0,C 180,E1 -4371.53,E2 -4371.53} C_VEL
LIN {X 0,Y 530.975,Z 117.154,A -85,B 0,C 180,E1 -4374.382,E2 -4374.382} C_VEL
LIN {X 0,Y 530.965,Z 117.154,A -85,B 0,C 180,E1 -4377.134,E2 -4377.134} C_VEL
LIN {X 0,Y 530.969,Z 117.16,A -85,B 0,C 180,E1 -4379.803,E2 -4379.803} C_VEL
LIN {X 0,Y 531.012,Z 117.147,A -85,B 0,C 180,E1 -4382.468,E2 -4382.468} C_VEL
LIN {X 0,Y 531.003,Z 117.151,A -85,B 0,C 180,E1 -4384.943,E2 -4384.943} C_VEL
LIN {X 0,Y 531.028,Z 117.279,A -85,B 0,C 180,E1 -4388.185,E2 -4388.185} C_VEL
LIN {X 0,Y 531.698,Z 121.724,A -85,B 0,C 180,E1 -4389.091,E2 -4389.091} C_VEL
LIN {X 0,Y 531.363,Z 138.274,A -85,B 0,C 180,E1 -4392.231,E2 -4392.231} C_VEL
LIN {X 0,Y 531.073,Z 153.86,A -85,B 0,C 180,E1 -4395.147,E2 -4395.147} C_VEL
LIN {X 0,Y 530.897,Z 170.552,A -85,B 0,C 180,E1 -4398.208,E2 -4398.208} C_VEL
LIN {X 0,Y 531.221,Z 173.755,A -85,B 0,C 180,E1 -4398.302,E2 -4398.302} C_VEL
LIN {X 0,Y 531.896,Z 180.927,A -85,B 0,C 180,E1 -4398.413,E2 -4398.413} C_VEL
LIN {X 0,Y 531.75,Z 246.618,A -85,B 0,C 180,E1 -4399.313,E2 -4399.313} C_VEL
LIN {X 0,Y 531.628,Z 255.888,A -85,B 0,C 180,E1 -4399.527,E2 -4399.527} C_VEL
LIN {X 0,Y 531.492,Z 264.365,A -85,B 0,C 180,E1 -4399.813,E2 -4399.813} C_VEL
LIN {X 0,Y 531.39,Z 272.879,A -85,B 0,C 180,E1 -4400.196,E2 -4400.196} C_VEL
LIN {X 0,Y 531.235,Z 281.222,A -85,B 0,C 180,E1 -4400.674,E2 -4400.674} C_VEL
LIN {X 0,Y 531.076,Z 289.272,A -85,B 0,C 180,E1 -4401.247,E2 -4401.247} C_VEL
LIN {X 0,Y 530.899,Z 297.96,A -85,B 0,C 180,E1 -4402.01,E2 -4402.01} C_VEL
LIN {X 0,Y 530.766,Z 306.485,A -85,B 0,C 180,E1 -4402.965,E2 -4402.965} C_VEL
LIN {X 0,Y 530.693,Z 313.174,A -85,B 0,C 180,E1 -4403.919,E2 -4403.919} C_VEL
LIN {X 0,Y 530.541,Z 317.563,A -85,B 0,C 180,E1 -4404.68,E2 -4404.68} C_VEL
LIN {X 0,Y 530.544,Z 322.74,A -85,B 0,C 180,E1 -4405.822,E2 -4405.822} C_VEL
LIN {X 0,Y 530.469,Z 326.539,A -85,B 0,C 180,E1 -4406.962,E2 -4406.962} C_VEL
LIN {X 0,Y 530.412,Z 328.286,A -85,B 0,C 180,E1 -4407.722,E2 -4407.722} C_VEL
LIN {X 0,Y 530.359,Z 329.537,A -85,B 0,C 180,E1 -4408.482,E2 -4408.482} C_VEL
LIN {X 0,Y 530.342,Z 330.317,A -85,B 0,C 180,E1 -4409.241,E2 -4409.241} C_VEL
LIN {X 0,Y 530.343,Z 330.612,A -85,B 0,C 180,E1 -4410,E2 -4410} C_VEL
LIN {X 0,Y 530.342,Z 330.316,A -85,B 0,C 180,E1 -4410.759,E2 -4410.759} C_VEL
LIN {X 0,Y 530.359,Z 329.536,A -85,B 0,C 180,E1 -4411.519,E2 -4411.519} C_VEL
LIN {X 0,Y 530.412,Z 328.284,A -85,B 0,C 180,E1 -4412.278,E2 -4412.278} C_VEL
LIN {X 0,Y 530.494,Z 325.383,A -85,B 0,C 180,E1 -4413.418,E2 -4413.418} C_VEL
LIN {X 0,Y 530.544,Z 322.738,A -85,B 0,C 180,E1 -4414.178,E2 -4414.178} C_VEL
LIN {X 0,Y 530.542,Z 317.558,A -85,B 0,C 180,E1 -4415.321,E2 -4415.321} C_VEL
LIN {X 0,Y 530.685,Z 310.926,A -85,B 0,C 180,E1 -4416.437,E2 -4416.437} C_VEL
LIN {X 0,Y 530.782,Z 303.276,A -85,B 0,C 180,E1 -4417.418,E2 -4417.418} C_VEL
LIN {X 0,Y 530.953,Z 295.918,A -85,B 0,C 180,E1 -4418.181,E2 -4418.181} C_VEL
LIN {X 0,Y 531.107,Z 288.04,A -85,B 0,C 180,E1 -4418.849,E2 -4418.849} C_VEL
LIN {X 0,Y 531.27,Z 279.715,A -85,B 0,C 180,E1 -4419.422,E2 -4419.422} C_VEL
LIN {X 0,Y 531.455,Z 269.089,A -85,B 0,C 180,E1 -4419.995,E2 -4419.995} C_VEL
LIN {X 0,Y 531.586,Z 257.542,A -85,B 0,C 180,E1 -4420.426,E2 -4420.426} C_VEL
LIN {X 0,Y 531.749,Z 247.896,A -85,B 0,C 180,E1 -4420.663,E2 -4420.663} C_VEL
LIN {X 0,Y 531.797,Z 178.177,A -85,B 0,C 180,E1 -4421.626,E2 -4421.626} C_VEL
LIN {X 0,Y 530.882,Z 170.749,A -85,B 0,C 180,E1 -4421.774,E2 -4421.774} C_VEL
LIN {X 0,Y 531.064,Z 156.468,A -85,B 0,C 180,E1 -4424.367,E2 -4424.367} C_VEL
LIN {X 0,Y 531.334,Z 139.632,A -85,B 0,C 180,E1 -4427.513,E2 -4427.513} C_VEL
LIN {X 0,Y 531.629,Z 123.834,A -85,B 0,C 180,E1 -4430.507,E2 -4430.507} C_VEL
LIN {X 0,Y 531.428,Z 119.605,A -85,B 0,C 180,E1 -4431.327,E2 -4431.327} C_VEL
LIN {X 0,Y 530.994,Z 117.184,A -85,B 0,C 180,E1 -4431.865,E2 -4431.865} C_VEL
LIN {X 0,Y 531,Z 117.151,A -85,B 0,C 180,E1 -4435.058,E2 -4435.058} C_VEL
LIN {X 0,Y 531.014,Z 117.147,A -85,B 0,C 180,E1 -4437.596,E2 -4437.596} C_VEL
LIN {X 0,Y 530.975,Z 117.156,A -85,B 0,C 180,E1 -4440.645,E2 -4440.645} C_VEL
LIN {X 0,Y 530.988,Z 117.154,A -85,B 0,C 180,E1 -4443.773,E2 -4443.773} C_VEL
LIN {X 0,Y 530.955,Z 117.157,A -85,B 0,C 180,E1 -4446.559,E2 -4446.559} C_VEL
LIN {X 0,Y 530.986,Z 117.153,A -85,B 0,C 180,E1 -4449.444,E2 -4449.444} C_VEL
LIN {X 0,Y 530.978,Z 117.153,A -85,B 0,C 180,E1 -4452.457,E2 -4452.457} C_VEL
LIN {X 0,Y 530.976,Z 117.159,A -85,B 0,C 180,E1 -4455.622,E2 -4455.622} C_VEL
LIN {X 0,Y 530.997,Z 117.149,A -85,B 0,C 180,E1 -4458.565,E2 -4458.565} C_VEL
LIN {X 0,Y 530.958,Z 117.163,A -85,B 0,C 180,E1 -4461.529,E2 -4461.529} C_VEL
LIN {X 0,Y 530.978,Z 117.152,A -85,B 0,C 180,E1 -4464.382,E2 -4464.382} C_VEL
LIN {X 0,Y 530.968,Z 117.159,A -85,B 0,C 180,E1 -4467.134,E2 -4467.134} C_VEL
LIN {X 0,Y 530.97,Z 117.154,A -85,B 0,C 180,E1 -4469.803,E2 -4469.803} C_VEL
LIN {X 0,Y 531.014,Z 117.148,A -85,B 0,C 180,E1 -4472.468,E2 -4472.468} C_VEL
LIN {X 0,Y 531.006,Z 117.156,A -85,B 0,C 180,E1 -4474.943,E2 -4474.943} C_VEL
LIN {X 0,Y 530.973,Z 117.153,A -85,B 0,C 180,E1 -4478.247,E2 -4478.247} C_VEL
LIN {X 0,Y 530.997,Z 117.156,A -85,B 0,C 180,E1 -4480.677,E2 -4480.677} C_VEL
LIN {X 0,Y 530.987,Z 117.154,A -85,B 0,C 180,E1 -4483.071,E2 -4483.071} C_VEL
LIN {X 0,Y 531.021,Z 117.147,A -85,B 0,C 180,E1 -4485.436,E2 -4485.436} C_VEL
LIN {X 0,Y 531.038,Z 117.153,A -85,B 0,C 180,E1 -4488.55,E2 -4488.55} C_VEL
LIN {X 0,Y 531.056,Z 117.142,A -85,B 0,C 180,E1 -4491.63,E2 -4491.63} C_VEL
LIN {X 0,Y 531.12,Z 117.137,A -85,B 0,C 180,E1 -4494.685,E2 -4494.685} C_VEL
LIN {X 0,Y 531.14,Z 117.134,A -85,B 0,C 180,E1 -4497.725,E2 -4497.725} C_VEL
LIN {X 0,Y 531.154,Z 117.13,A -85,B 0,C 180,E1 -4500.758,E2 -4500.758} C_VEL
LIN {X 0,Y 531.104,Z 117.136,A -85,B 0,C 180,E1 -4503.034,E2 -4503.034} C_VEL
LIN {X 0,Y 531.085,Z 117.144,A -85,B 0,C 180,E1 -4506.077,E2 -4506.077} C_VEL
LIN {X 0,Y 531.03,Z 117.147,A -85,B 0,C 180,E1 -4509.138,E2 -4509.138} C_VEL
LIN {X 0,Y 531.042,Z 117.145,A -85,B 0,C 180,E1 -4512.225,E2 -4512.225} C_VEL
LIN {X 0,Y 530.998,Z 117.156,A -85,B 0,C 180,E1 -4515.35,E2 -4515.35} C_VEL
LIN {X 0,Y 530.99,Z 117.15,A -85,B 0,C 180,E1 -4518.521,E2 -4518.521} C_VEL
LIN {X 0,Y 531.001,Z 117.153,A -85,B 0,C 180,E1 -4520.938,E2 -4520.938} C_VEL
LIN {X 0,Y 530.967,Z 117.153,A -85,B 0,C 180,E1 -4524.225,E2 -4524.225} C_VEL
LIN {X 0,Y 531.003,Z 117.153,A -85,B 0,C 180,E1 -4526.744,E2 -4526.744} C_VEL
LIN {X 0,Y 530.984,Z 117.155,A -85,B 0,C 180,E1 -4529.323,E2 -4529.323} C_VEL
LIN {X 0,Y 530.967,Z 117.153,A -85,B 0,C 180,E1 -4532.1,E2 -4532.1} C_VEL
LIN {X 0,Y 530.986,Z 117.158,A -85,B 0,C 180,E1 -4534.853,E2 -4534.853} C_VEL
LIN {X 0,Y 530.968,Z 117.153,A -85,B 0,C 180,E1 -4537.508,E2 -4537.508} C_VEL
LIN {X 0,Y 530.982,Z 117.158,A -85,B 0,C 180,E1 -4540.433,E2 -4540.433} C_VEL
LIN {X 0,Y 530.962,Z 117.154,A -85,B 0,C 180,E1 -4543.281,E2 -4543.281} C_VEL
LIN {X 0,Y 530.953,Z 117.155,A -85,B 0,C 180,E1 -4543.56,E2 -4543.56} C_VEL
LIN {X 0,Y 530.28,Z 117.246,A -85,B 0,C 180,E1 -4544.193,E2 -4544.193} C_VEL
LIN {X 0,Y 527.433,Z 117.599,A -85,B 0,C 180,E1 -4545.222,E2 -4545.222} C_VEL
LIN {X 0,Y 525.032,Z 117.898,A -85,B 0,C 180,E1 -4546.051,E2 -4546.051} C_VEL
LIN {X 0,Y 524,Z 118.025,A -85,B 0,C 180,E1 -4546.69,E2 -4546.69} C_VEL
LIN {X 0,Y 523.916,Z 118.033,A -85,B 0,C 180,E1 -4546.907,E2 -4546.907} C_VEL
LIN {X 0,Y 523.95,Z 118.032,A -85,B 0,C 180,E1 -4549.921,E2 -4549.921} C_VEL
LIN {X 0,Y 523.912,Z 118.032,A -85,B 0,C 180,E1 -4552.868,E2 -4552.868} C_VEL
LIN {X 0,Y 523.931,Z 118.034,A -85,B 0,C 180,E1 -4555.71,E2 -4555.71} C_VEL
LIN {X 0,Y 523.922,Z 118.032,A -85,B 0,C 180,E1 -4558.456,E2 -4558.456} C_VEL
LIN {X 0,Y 523.941,Z 118.029,A -85,B 0,C 180,E1 -4561.125,E2 -4561.125} C_VEL
LIN {X 0,Y 523.987,Z 118.027,A -85,B 0,C 180,E1 -4563.98,E2 -4563.98} C_VEL
LIN {X 0,Y 523.912,Z 118.036,A -85,B 0,C 180,E1 -4567.106,E2 -4567.106} C_VEL
LIN {X 0,Y 524.021,Z 118.024,A -85,B 0,C 180,E1 -4570.41,E2 -4570.41} C_VEL
LIN {X 0,Y 524.057,Z 118.368,A -85,B 0,C 180,E1 -4570.717,E2 -4570.717} C_VEL
LIN {X 0,Y 524.203,Z 126.373,A -85,B 0,C 180,E1 -4572.492,E2 -4572.492} C_VEL
LIN {X 0,Y 523.966,Z 140.849,A -85,B 0,C 180,E1 -4575.632,E2 -4575.632} C_VEL
LIN {X 0,Y 523.796,Z 152.715,A -85,B 0,C 180,E1 -4578.107,E2 -4578.107} C_VEL
LIN {X 0,Y 524.145,Z 155.144,A -85,B 0,C 180,E1 -4578.188,E2 -4578.188} C_VEL
LIN {X 0,Y 525.012,Z 162.502,A -85,B 0,C 180,E1 -4578.308,E2 -4578.308} C_VEL
LIN {X 0,Y 524.78,Z 228.023,A -85,B 0,C 180,E1 -4579.218,E2 -4579.218} C_VEL
LIN {X 0,Y 524.677,Z 237.219,A -85,B 0,C 180,E1 -4579.435,E2 -4579.435} C_VEL
LIN {X 0,Y 524.584,Z 246.859,A -85,B 0,C 180,E1 -4579.775,E2 -4579.775} C_VEL
LIN {X 0,Y 524.446,Z 255.06,A -85,B 0,C 180,E1 -4580.162,E2 -4580.162} C_VEL
LIN {X 0,Y 524.253,Z 264.68,A -85,B 0,C 180,E1 -4580.742,E2 -4580.742} C_VEL
LIN {X 0,Y 524.01,Z 274.519,A -85,B 0,C 180,E1 -4581.516,E2 -4581.516} C_VEL
LIN {X 0,Y 523.84,Z 282.266,A -85,B 0,C 180,E1 -4582.29,E2 -4582.29} C_VEL
LIN {X 0,Y 523.708,Z 288.635,A -85,B 0,C 180,E1 -4583.063,E2 -4583.063} C_VEL
LIN {X 0,Y 523.724,Z 293.926,A -85,B 0,C 180,E1 -4583.837,E2 -4583.837} C_VEL
LIN {X 0,Y 523.488,Z 298.35,A -85,B 0,C 180,E1 -4584.607,E2 -4584.607} C_VEL
LIN {X 0,Y 523.495,Z 303.543,A -85,B 0,C 180,E1 -4585.765,E2 -4585.765} C_VEL
LIN {X 0,Y 523.442,Z 306.215,A -85,B 0,C 180,E1 -4586.536,E2 -4586.536} C_VEL
LIN {X 0,Y 523.338,Z 309.14,A -85,B 0,C 180,E1 -4587.691,E2 -4587.691} C_VEL
LIN {X 0,Y 523.274,Z 310.424,A -85,B 0,C 180,E1 -4588.461,E2 -4588.461} C_VEL
LIN {X 0,Y 523.249,Z 311.238,A -85,B 0,C 180,E1 -4589.23,E2 -4589.23} C_VEL
LIN {X 0,Y 523.248,Z 311.547,A -85,B 0,C 180,E1 -4590,E2 -4590} C_VEL
LIN {X 0,Y 523.25,Z 311.275,A -85,B 0,C 180,E1 -4590.769,E2 -4590.769} C_VEL
LIN {X 0,Y 523.275,Z 310.538,A -85,B 0,C 180,E1 -4591.539,E2 -4591.539} C_VEL
LIN {X 0,Y 523.338,Z 309.331,A -85,B 0,C 180,E1 -4592.309,E2 -4592.309} C_VEL
LIN {X 0,Y 523.427,Z 306.485,A -85,B 0,C 180,E1 -4593.464,E2 -4593.464} C_VEL
LIN {X 0,Y 523.491,Z 303.898,A -85,B 0,C 180,E1 -4594.234,E2 -4594.234} C_VEL
LIN {X 0,Y 523.484,Z 298.799,A -85,B 0,C 180,E1 -4595.392,E2 -4595.392} C_VEL
LIN {X 0,Y 523.735,Z 293.452,A -85,B 0,C 180,E1 -4596.332,E2 -4596.332} C_VEL
LIN {X 0,Y 523.763,Z 286.426,A -85,B 0,C 180,E1 -4597.323,E2 -4597.323} C_VEL
LIN {X 0,Y 523.97,Z 277.499,A -85,B 0,C 180,E1 -4598.29,E2 -4598.29} C_VEL
LIN {X 0,Y 524.167,Z 269.748,A -85,B 0,C 180,E1 -4598.967,E2 -4598.967} C_VEL
LIN {X 0,Y 524.282,Z 261.577,A -85,B 0,C 180,E1 -4599.549,E2 -4599.549} C_VEL
LIN {X 0,Y 524.481,Z 253.052,A -85,B 0,C 180,E1 -4600.032,E2 -4600.032} C_VEL
LIN {X 0,Y 524.669,Z 241.802,A -85,B 0,C 180,E1 -4600.516,E2 -4600.516} C_VEL
LIN {X 0,Y 524.844,Z 230.227,A -85,B 0,C 180,E1 -4600.829,E2 -4600.829} C_VEL
LIN {X 0,Y 524.884,Z 205.6,A -85,B 0,C 180,E1 -4601.195,E2 -4601.195} C_VEL
LIN {X 0,Y 524.815,Z 159.705,A -85,B 0,C 180,E1 -4601.824,E2 -4601.824} C_VEL
LIN {X 0,Y 523.866,Z 153.217,A -85,B 0,C 180,E1 -4601.947,E2 -4601.947} C_VEL
LIN {X 0,Y 523.807,Z 151.934,A -85,B 0,C 180,E1 -4602.102,E2 -4602.102} C_VEL
LIN {X 0,Y 523.998,Z 137.353,A -85,B 0,C 180,E1 -4605.21,E2 -4605.21} C_VEL
LIN {X 0,Y 524.265,Z 122.894,A -85,B 0,C 180,E1 -4608.362,E2 -4608.362} C_VEL
LIN {X 0,Y 524.053,Z 118.122,A -85,B 0,C 180,E1 -4609.461,E2 -4609.461} C_VEL
LIN {X 0,Y 523.92,Z 118.038,A -85,B 0,C 180,E1 -4612.243,E2 -4612.243} C_VEL
LIN {X 0,Y 523.947,Z 118.027,A -85,B 0,C 180,E1 -4615.419,E2 -4615.419} C_VEL
LIN {X 0,Y 523.969,Z 118.029,A -85,B 0,C 180,E1 -4617.999,E2 -4617.999} C_VEL
LIN {X 0,Y 523.945,Z 118.029,A -85,B 0,C 180,E1 -4620.854,E2 -4620.854} C_VEL
LIN {X 0,Y 523.933,Z 118.033,A -85,B 0,C 180,E1 -4623.73,E2 -4623.73} C_VEL
LIN {X 0,Y 523.919,Z 118.035,A -85,B 0,C 180,E1 -4626.403,E2 -4626.403} C_VEL
LIN {X 0,Y 523.92,Z 118.031,A -85,B 0,C 180,E1 -4629.084,E2 -4629.084} C_VEL
LIN {X 0,Y 523.951,Z 118.031,A -85,B 0,C 180,E1 -4632.119,E2 -4632.119} C_VEL
LIN {X 0,Y 523.943,Z 118.032,A -85,B 0,C 180,E1 -4635.31,E2 -4635.31} C_VEL
LIN {X 0,Y 523.957,Z 118.026,A -85,B 0,C 180,E1 -4638.689,E2 -4638.689} C_VEL
